      ON    I      7.7;
      O     ;
      A     M     61.5;
      AN    I      0.1;
      =     M     61.5;
NETWORK
TITLE =PROFINET ALARM-모듈이상이나 통신케이블단선(1~10)
//
//
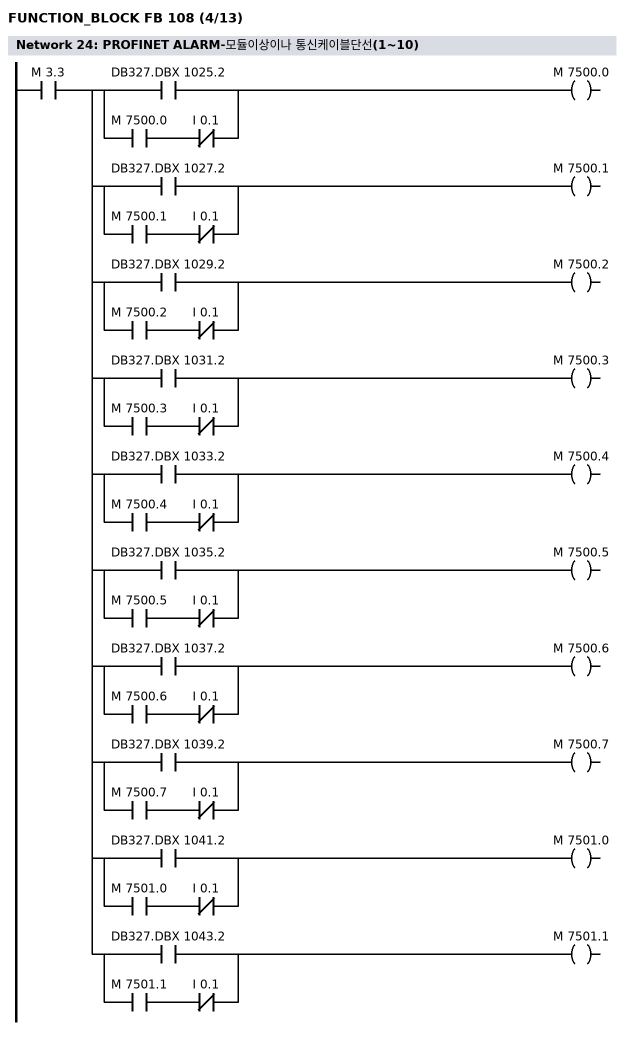
      A     M      3.3;
      =     L      0.0;
      A     L      0.0;
      A(    ;
      O     DB327.DBX 1025.2;
      O     ;
      A     M   7500.0;
      AN    I      0.1;
      )     ;
      =     M   7500.0;
      A     L      0.0;
      A(    ;
      O     DB327.DBX 1027.2;
      O     ;
      A     M   7500.1;
      AN    I      0.1;
      )     ;
      =     M   7500.1;
      A     L      0.0;
      A(    ;
      O     DB327.DBX 1029.2;
      O     ;
      A     M   7500.2;
      AN    I      0.1;
      )     ;
      =     M   7500.2;
      A     L      0.0;
      A(    ;
      O     DB327.DBX 1031.2;
      O     ;
      A     M   7500.3;
      AN    I      0.1;
      )     ;
      =     M   7500.3;
      A     L      0.0;
      A(    ;
      O     DB327.DBX 1033.2;
      O     ;
      A     M   7500.4;
      AN    I      0.1;
      )     ;
      =     M   7500.4;
      A     L      0.0;
      A(    ;
      O     DB327.DBX 1035.2;
      O     ;
      A     M   7500.5;
      AN    I      0.1;
      )     ;
      =     M   7500.5;
      A     L      0.0;
      A(    ;
      O     DB327.DBX 1037.2;
      O     ;
      A     M   7500.6;
      AN    I      0.1;
      )     ;
      =     M   7500.6;
      A     L      0.0;
      A(    ;
      O     DB327.DBX 1039.2;
      O     ;
      A     M   7500.7;
      AN    I      0.1;
      )     ;
      =     M   7500.7;
      A     L      0.0;
      A(    ;
      O     DB327.DBX 1041.2;
      O     ;
      A     M   7501.0;
      AN    I      0.1;
      )     ;
      =     M   7501.0;
      A     L      0.0;
      A(    ;
      O     DB327.DBX 1043.2;
      O     ;
      A     M   7501.1;
      AN    I      0.1;
      )     ;
      =     M   7501.1;
NETWORK
TITLE =PROFINET ALARM-모듈이상이나 통신케이블단선(11~20)
//
//
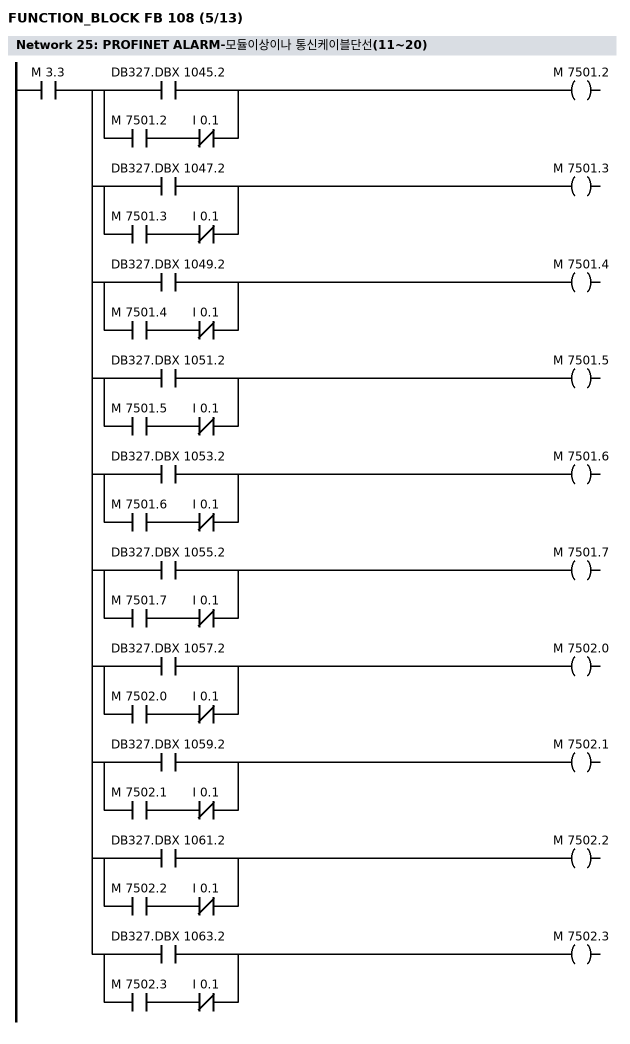
      A     M      3.3;
      =     L      0.0;
      A     L      0.0;
      A(    ;
      O     DB327.DBX 1045.2;
      O     ;
      A     M   7501.2;
      AN    I      0.1;
      )     ;
      =     M   7501.2;
      A     L      0.0;
      A(    ;
      O     DB327.DBX 1047.2;
      O     ;
      A     M   7501.3;
      AN    I      0.1;
      )     ;
      =     M   7501.3;
      A     L      0.0;
      A(    ;
      O     DB327.DBX 1049.2;
      O     ;
      A     M   7501.4;
      AN    I      0.1;
      )     ;
      =     M   7501.4;
      A     L      0.0;
      A(    ;
      O     DB327.DBX 1051.2;
      O     ;
      A     M   7501.5;
      AN    I      0.1;
      )     ;
      =     M   7501.5;
      A     L      0.0;
      A(    ;
      O     DB327.DBX 1053.2;
      O     ;
      A     M   7501.6;
      AN    I      0.1;
      )     ;
      =     M   7501.6;
      A     L      0.0;
      A(    ;
      O     DB327.DBX 1055.2;
      O     ;
      A     M   7501.7;
      AN    I      0.1;
      )     ;
      =     M   7501.7;
      A     L      0.0;
      A(    ;
      O     DB327.DBX 1057.2;
      O     ;
      A     M   7502.0;
      AN    I      0.1;
      )     ;
      =     M   7502.0;
      A     L      0.0;
      A(    ;
      O     DB327.DBX 1059.2;
      O     ;
      A     M   7502.1;
      AN    I      0.1;
      )     ;
      =     M   7502.1;
      A     L      0.0;
      A(    ;
      O     DB327.DBX 1061.2;
      O     ;
      A     M   7502.2;
      AN    I      0.1;
      )     ;
      =     M   7502.2;
      A     L      0.0;
      A(    ;
      O     DB327.DBX 1063.2;
      O     ;
      A     M   7502.3;
      AN    I      0.1;
      )     ;
      =     M   7502.3;
NETWORK
TITLE =PROFINET ALARM-모듈이상이나 통신케이블단선(21~30)
//
//
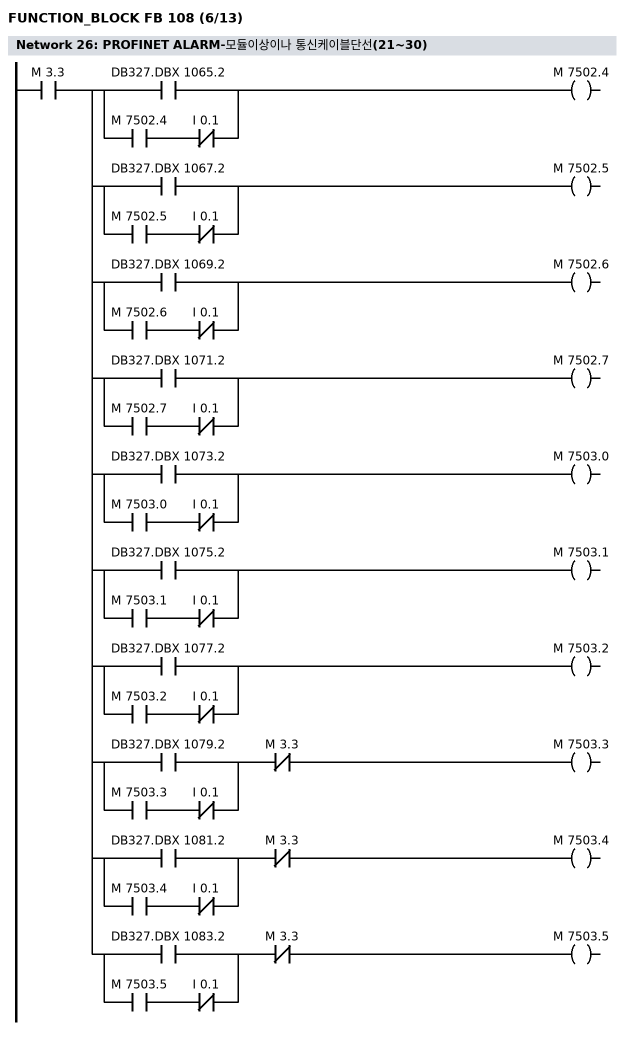
      A     M      3.3;
      =     L      0.0;
      A     L      0.0;
      A(    ;
      O     DB327.DBX 1065.2;
      O     ;
      A     M   7502.4;
      AN    I      0.1;
      )     ;
      =     M   7502.4;
      A     L      0.0;
      A(    ;
      O     DB327.DBX 1067.2;
      O     ;
      A     M   7502.5;
      AN    I      0.1;
      )     ;
      =     M   7502.5;
      A     L      0.0;
      A(    ;
      O     DB327.DBX 1069.2;
      O     ;
      A     M   7502.6;
      AN    I      0.1;
      )     ;
      =     M   7502.6;
      A     L      0.0;
      A(    ;
      O     DB327.DBX 1071.2;
      O     ;
      A     M   7502.7;
      AN    I      0.1;
      )     ;
      =     M   7502.7;
      A     L      0.0;
      A(    ;
      O     DB327.DBX 1073.2;
      O     ;
      A     M   7503.0;
      AN    I      0.1;
      )     ;
      =     M   7503.0;
      A     L      0.0;
      A(    ;
      O     DB327.DBX 1075.2;
      O     ;
      A     M   7503.1;
      AN    I      0.1;
      )     ;
      =     M   7503.1;
      A     L      0.0;
      A(    ;
      O     DB327.DBX 1077.2;
      O     ;
      A     M   7503.2;
      AN    I      0.1;
      )     ;
      =     M   7503.2;
      A     L      0.0;
      A(    ;
      O     DB327.DBX 1079.2;
      O     ;
      A     M   7503.3;
      AN    I      0.1;
      )     ;
      AN    M      3.3;
      =     M   7503.3;
      A     L      0.0;
      A(    ;
      O     DB327.DBX 1081.2;
      O     ;
      A     M   7503.4;
      AN    I      0.1;
      )     ;
      AN    M      3.3;
      =     M   7503.4;
      A     L      0.0;
      A(    ;
      O     DB327.DBX 1083.2;
      O     ;
      A     M   7503.5;
      AN    I      0.1;
      )     ;
      AN    M      3.3;
      =     M   7503.5;
NETWORK
TITLE =PROFINET ALARM-모듈이상이나 통신케이블단선(31~40)
//
//
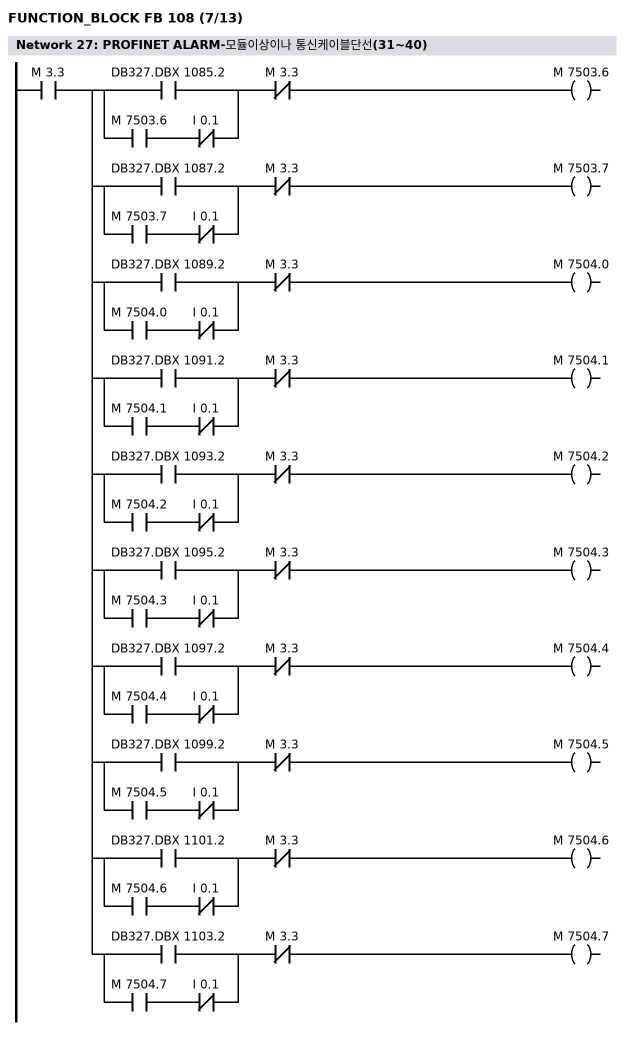
      A     M      3.3;
      =     L      0.0;
      A     L      0.0;
      A(    ;
      O     DB327.DBX 1085.2;
      O     ;
      A     M   7503.6;
      AN    I      0.1;
      )     ;
      AN    M      3.3;
      =     M   7503.6;
      A     L      0.0;
      A(    ;
      O     DB327.DBX 1087.2;
      O     ;
      A     M   7503.7;
      AN    I      0.1;
      )     ;
      AN    M      3.3;
      =     M   7503.7;
      A     L      0.0;
      A(    ;
      O     DB327.DBX 1089.2;
      O     ;
      A     M   7504.0;
      AN    I      0.1;
      )     ;
      AN    M      3.3;
      =     M   7504.0;
      A     L      0.0;
      A(    ;
      O     DB327.DBX 1091.2;
      O     ;
      A     M   7504.1;
      AN    I      0.1;
      )     ;
      AN    M      3.3;
      =     M   7504.1;
      A     L      0.0;
      A(    ;
      O     DB327.DBX 1093.2;
      O     ;
      A     M   7504.2;
      AN    I      0.1;
      )     ;
      AN    M      3.3;
      =     M   7504.2;
      A     L      0.0;
      A(    ;
      O     DB327.DBX 1095.2;
      O     ;
      A     M   7504.3;
      AN    I      0.1;
      )     ;
      AN    M      3.3;
      =     M   7504.3;
      A     L      0.0;
      A(    ;
      O     DB327.DBX 1097.2;
      O     ;
      A     M   7504.4;
      AN    I      0.1;
      )     ;
      AN    M      3.3;
      =     M   7504.4;
      A     L      0.0;
      A(    ;
      O     DB327.DBX 1099.2;
      O     ;
      A     M   7504.5;
      AN    I      0.1;
      )     ;
      AN    M      3.3;
      =     M   7504.5;
      A     L      0.0;
      A(    ;
      O     DB327.DBX 1101.2;
      O     ;
      A     M   7504.6;
      AN    I      0.1;
      )     ;
      AN    M      3.3;
      =     M   7504.6;
      A     L      0.0;
      A(    ;
      O     DB327.DBX 1103.2;
      O     ;
      A     M   7504.7;
      AN    I      0.1;
      )     ;
      AN    M      3.3;
      =     M   7504.7;
NETWORK
TITLE =PROFINET ALARM-모듈이상이나 통신케이블단선(150~159)
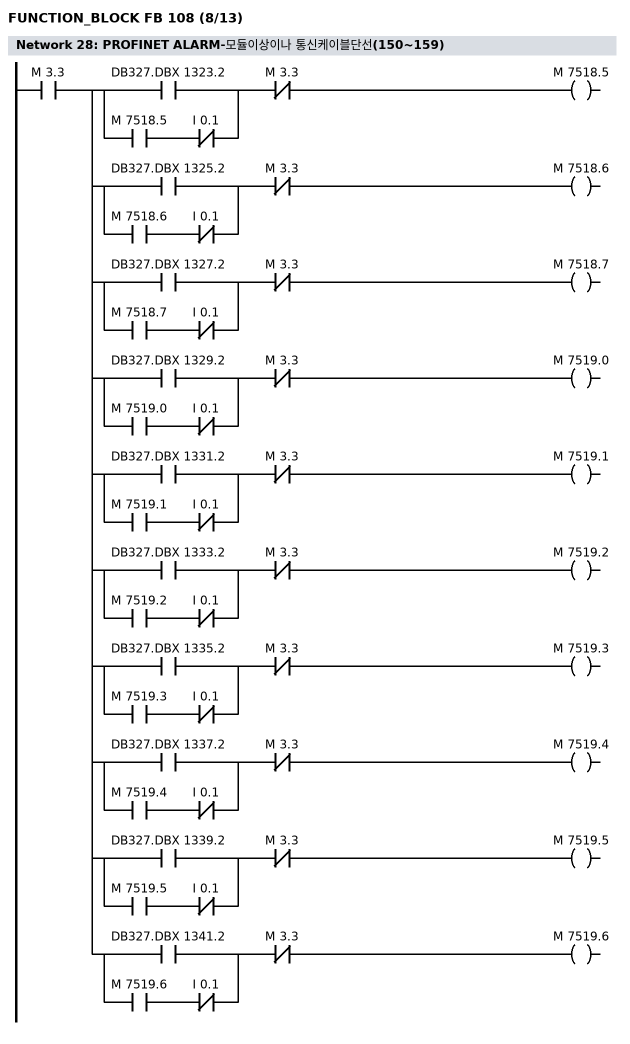

      A     M      3.3;
      =     L      0.0;
      A     L      0.0;
      A(    ;
      O     DB327.DBX 1323.2;
      O     ;
      A     M   7518.5;
      AN    I      0.1;
      )     ;
      AN    M      3.3;
      =     M   7518.5;
      A     L      0.0;
      A(    ;
      O     DB327.DBX 1325.2;
      O     ;
      A     M   7518.6;
      AN    I      0.1;
      )     ;
      AN    M      3.3;
      =     M   7518.6;
      A     L      0.0;
      A(    ;
      O     DB327.DBX 1327.2;
      O     ;
      A     M   7518.7;
      AN    I      0.1;
      )     ;
      AN    M      3.3;
      =     M   7518.7;
      A     L      0.0;
      A(    ;
      O     DB327.DBX 1329.2;
      O     ;
      A     M   7519.0;
      AN    I      0.1;
      )     ;
      AN    M      3.3;
      =     M   7519.0;
      A     L      0.0;
      A(    ;
      O     DB327.DBX 1331.2;
      O     ;
      A     M   7519.1;
      AN    I      0.1;
      )     ;
      AN    M      3.3;
      =     M   7519.1;
      A     L      0.0;
      A(    ;
      O     DB327.DBX 1333.2;
      O     ;
      A     M   7519.2;
      AN    I      0.1;
      )     ;
      AN    M      3.3;
      =     M   7519.2;
      A     L      0.0;
      A(    ;
      O     DB327.DBX 1335.2;
      O     ;
      A     M   7519.3;
      AN    I      0.1;
      )     ;
      AN    M      3.3;
      =     M   7519.3;
      A     L      0.0;
      A(    ;
      O     DB327.DBX 1337.2;
      O     ;
      A     M   7519.4;
      AN    I      0.1;
      )     ;
      AN    M      3.3;
      =     M   7519.4;
      A     L      0.0;
      A(    ;
      O     DB327.DBX 1339.2;
      O     ;
      A     M   7519.5;
      AN    I      0.1;
      )     ;
      AN    M      3.3;
      =     M   7519.5;
      A     L      0.0;
      A(    ;
      O     DB327.DBX 1341.2;
      O     ;
      A     M   7519.6;
      AN    I      0.1;
      )     ;
      AN    M      3.3;
      =     M   7519.6;
NETWORK
TITLE =PROFINET MODULE ERROR(1~10)
//
//
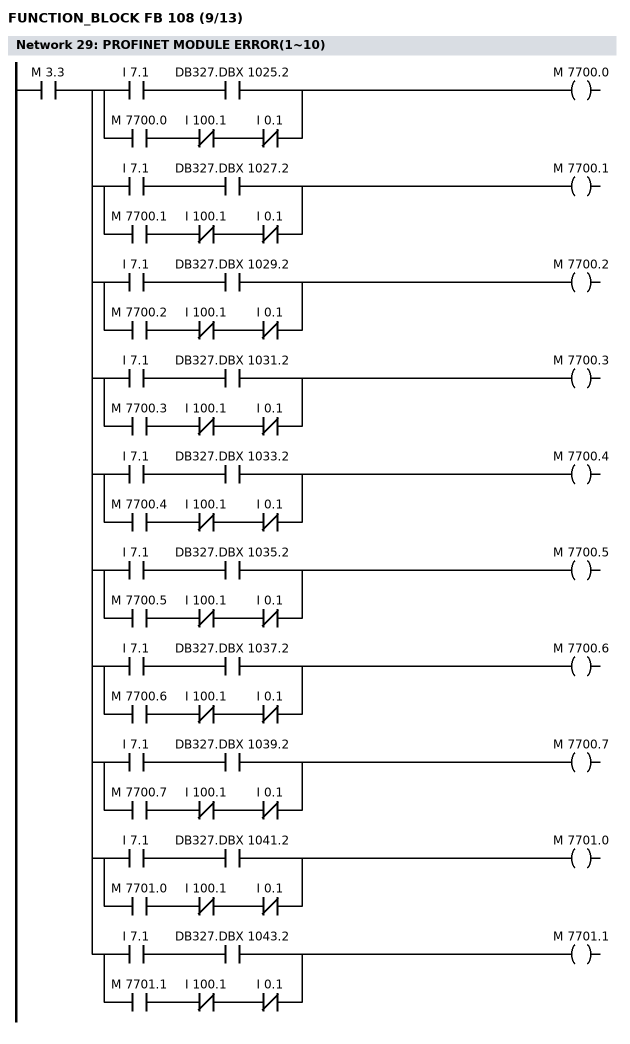
      A     M      3.3;
      =     L      0.0;
      A     L      0.0;
      A(    ;
      A     I      7.1;
      A     DB327.DBX 1025.2;
      O     ;
      A     M   7700.0;
      AN    I    100.1;
      AN    I      0.1;
      )     ;
      =     M   7700.0;
      A     L      0.0;
      A(    ;
      A     I      7.1;
      A     DB327.DBX 1027.2;
      O     ;
      A     M   7700.1;
      AN    I    100.1;
      AN    I      0.1;
      )     ;
      =     M   7700.1;
      A     L      0.0;
      A(    ;
      A     I      7.1;
      A     DB327.DBX 1029.2;
      O     ;
      A     M   7700.2;
      AN    I    100.1;
      AN    I      0.1;
      )     ;
      =     M   7700.2;
      A     L      0.0;
      A(    ;
      A     I      7.1;
      A     DB327.DBX 1031.2;
      O     ;
      A     M   7700.3;
      AN    I    100.1;
      AN    I      0.1;
      )     ;
      =     M   7700.3;
      A     L      0.0;
      A(    ;
      A     I      7.1;
      A     DB327.DBX 1033.2;
      O     ;
      A     M   7700.4;
      AN    I    100.1;
      AN    I      0.1;
      )     ;
      =     M   7700.4;
      A     L      0.0;
      A(    ;
      A     I      7.1;
      A     DB327.DBX 1035.2;
      O     ;
      A     M   7700.5;
      AN    I    100.1;
      AN    I      0.1;
      )     ;
      =     M   7700.5;
      A     L      0.0;
      A(    ;
      A     I      7.1;
      A     DB327.DBX 1037.2;
      O     ;
      A     M   7700.6;
      AN    I    100.1;
      AN    I      0.1;
      )     ;
      =     M   7700.6;
      A     L      0.0;
      A(    ;
      A     I      7.1;
      A     DB327.DBX 1039.2;
      O     ;
      A     M   7700.7;
      AN    I    100.1;
      AN    I      0.1;
      )     ;
      =     M   7700.7;
      A     L      0.0;
      A(    ;
      A     I      7.1;
      A     DB327.DBX 1041.2;
      O     ;
      A     M   7701.0;
      AN    I    100.1;
      AN    I      0.1;
      )     ;
      =     M   7701.0;
      A     L      0.0;
      A(    ;
      A     I      7.1;
      A     DB327.DBX 1043.2;
      O     ;
      A     M   7701.1;
      AN    I    100.1;
      AN    I      0.1;
      )     ;
      =     M   7701.1;
NETWORK
TITLE =PROFINET MODULE ERROR(11~20)
//
//
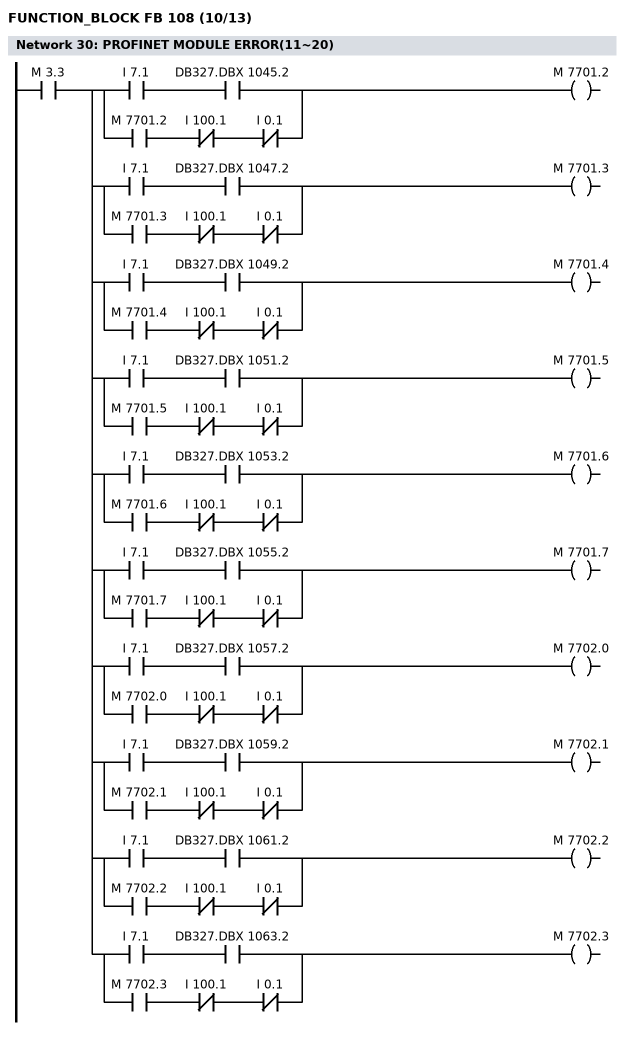
      A     M      3.3;
      =     L      0.0;
      A     L      0.0;
      A(    ;
      A     I      7.1;
      A     DB327.DBX 1045.2;
      O     ;
      A     M   7701.2;
      AN    I    100.1;
      AN    I      0.1;
      )     ;
      =     M   7701.2;
      A     L      0.0;
      A(    ;
      A     I      7.1;
      A     DB327.DBX 1047.2;
      O     ;
      A     M   7701.3;
      AN    I    100.1;
      AN    I      0.1;
      )     ;
      =     M   7701.3;
      A     L      0.0;
      A(    ;
      A     I      7.1;
      A     DB327.DBX 1049.2;
      O     ;
      A     M   7701.4;
      AN    I    100.1;
      AN    I      0.1;
      )     ;
      =     M   7701.4;
      A     L      0.0;
      A(    ;
      A     I      7.1;
      A     DB327.DBX 1051.2;
      O     ;
      A     M   7701.5;
      AN    I    100.1;
      AN    I      0.1;
      )     ;
      =     M   7701.5;
      A     L      0.0;
      A(    ;
      A     I      7.1;
      A     DB327.DBX 1053.2;
      O     ;
      A     M   7701.6;
      AN    I    100.1;
      AN    I      0.1;
      )     ;
      =     M   7701.6;
      A     L      0.0;
      A(    ;
      A     I      7.1;
      A     DB327.DBX 1055.2;
      O     ;
      A     M   7701.7;
      AN    I    100.1;
      AN    I      0.1;
      )     ;
      =     M   7701.7;
      A     L      0.0;
      A(    ;
      A     I      7.1;
      A     DB327.DBX 1057.2;
      O     ;
      A     M   7702.0;
      AN    I    100.1;
      AN    I      0.1;
      )     ;
      =     M   7702.0;
      A     L      0.0;
      A(    ;
      A     I      7.1;
      A     DB327.DBX 1059.2;
      O     ;
      A     M   7702.1;
      AN    I    100.1;
      AN    I      0.1;
      )     ;
      =     M   7702.1;
      A     L      0.0;
      A(    ;
      A     I      7.1;
      A     DB327.DBX 1061.2;
      O     ;
      A     M   7702.2;
      AN    I    100.1;
      AN    I      0.1;
      )     ;
      =     M   7702.2;
      A     L      0.0;
      A(    ;
      A     I      7.1;
      A     DB327.DBX 1063.2;
      O     ;
      A     M   7702.3;
      AN    I    100.1;
      AN    I      0.1;
      )     ;
      =     M   7702.3;
NETWORK
TITLE =PROFINET MODULE ERROR(21~30)
//
//
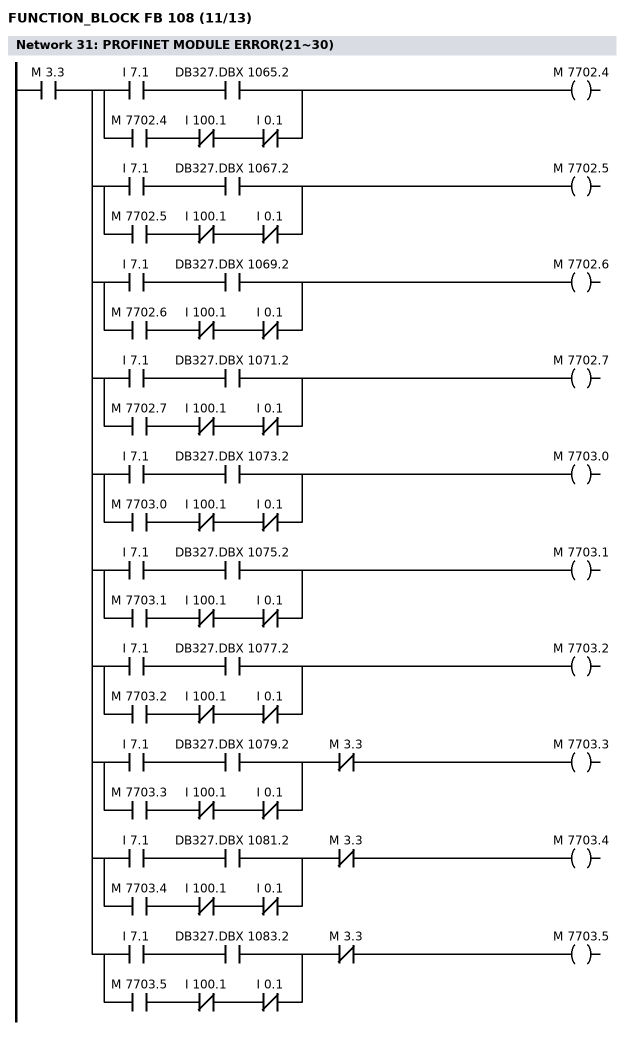
      A     M      3.3;
      =     L      0.0;
      A     L      0.0;
      A(    ;
      A     I      7.1;
      A     DB327.DBX 1065.2;
      O     ;
      A     M   7702.4;
      AN    I    100.1;
      AN    I      0.1;
      )     ;
      =     M   7702.4;
      A     L      0.0;
      A(    ;
      A     I      7.1;
      A     DB327.DBX 1067.2;
      O     ;
      A     M   7702.5;
      AN    I    100.1;
      AN    I      0.1;
      )     ;
      =     M   7702.5;
      A     L      0.0;
      A(    ;
      A     I      7.1;
      A     DB327.DBX 1069.2;
      O     ;
      A     M   7702.6;
      AN    I    100.1;
      AN    I      0.1;
      )     ;
      =     M   7702.6;
      A     L      0.0;
      A(    ;
      A     I      7.1;
      A     DB327.DBX 1071.2;
      O     ;
      A     M   7702.7;
      AN    I    100.1;
      AN    I      0.1;
      )     ;
      =     M   7702.7;
      A     L      0.0;
      A(    ;
      A     I      7.1;
      A     DB327.DBX 1073.2;
      O     ;
      A     M   7703.0;
      AN    I    100.1;
      AN    I      0.1;
      )     ;
      =     M   7703.0;
      A     L      0.0;
      A(    ;
      A     I      7.1;
      A     DB327.DBX 1075.2;
      O     ;
      A     M   7703.1;
      AN    I    100.1;
      AN    I      0.1;
      )     ;
      =     M   7703.1;
      A     L      0.0;
      A(    ;
      A     I      7.1;
      A     DB327.DBX 1077.2;
      O     ;
      A     M   7703.2;
      AN    I    100.1;
      AN    I      0.1;
      )     ;
      =     M   7703.2;
      A     L      0.0;
      A(    ;
      A     I      7.1;
      A     DB327.DBX 1079.2;
      O     ;
      A     M   7703.3;
      AN    I    100.1;
      AN    I      0.1;
      )     ;
      AN    M      3.3;
      =     M   7703.3;
      A     L      0.0;
      A(    ;
      A     I      7.1;
      A     DB327.DBX 1081.2;
      O     ;
      A     M   7703.4;
      AN    I    100.1;
      AN    I      0.1;
      )     ;
      AN    M      3.3;
      =     M   7703.4;
      A     L      0.0;
      A(    ;
      A     I      7.1;
      A     DB327.DBX 1083.2;
      O     ;
      A     M   7703.5;
      AN    I    100.1;
      AN    I      0.1;
      )     ;
      AN    M      3.3;
      =     M   7703.5;
NETWORK
TITLE =PROFINET MODULE ERROR(31~40)
//
//
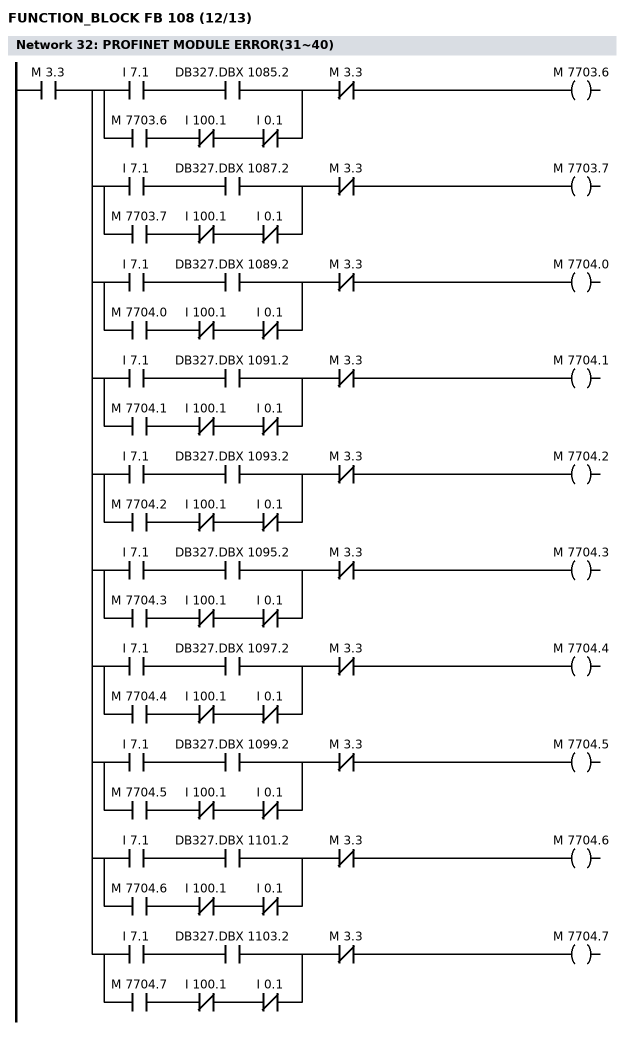
      A     M      3.3;
      =     L      0.0;
      A     L      0.0;
      A(    ;
      A     I      7.1;
      A     DB327.DBX 1085.2;
      O     ;
      A     M   7703.6;
      AN    I    100.1;
      AN    I      0.1;
      )     ;
      AN    M      3.3;
      =     M   7703.6;
      A     L      0.0;
      A(    ;
      A     I      7.1;
      A     DB327.DBX 1087.2;
      O     ;
      A     M   7703.7;
      AN    I    100.1;
      AN    I      0.1;
      )     ;
      AN    M      3.3;
      =     M   7703.7;
      A     L      0.0;
      A(    ;
      A     I      7.1;
      A     DB327.DBX 1089.2;
      O     ;
      A     M   7704.0;
      AN    I    100.1;
      AN    I      0.1;
      )     ;
      AN    M      3.3;
      =     M   7704.0;
      A     L      0.0;
      A(    ;
      A     I      7.1;
      A     DB327.DBX 1091.2;
      O     ;
      A     M   7704.1;
      AN    I    100.1;
      AN    I      0.1;
      )     ;
      AN    M      3.3;
      =     M   7704.1;
      A     L      0.0;
      A(    ;
      A     I      7.1;
      A     DB327.DBX 1093.2;
      O     ;
      A     M   7704.2;
      AN    I    100.1;
      AN    I      0.1;
      )     ;
      AN    M      3.3;
      =     M   7704.2;
      A     L      0.0;
      A(    ;
      A     I      7.1;
      A     DB327.DBX 1095.2;
      O     ;
      A     M   7704.3;
      AN    I    100.1;
      AN    I      0.1;
      )     ;
      AN    M      3.3;
      =     M   7704.3;
      A     L      0.0;
      A(    ;
      A     I      7.1;
      A     DB327.DBX 1097.2;
      O     ;
      A     M   7704.4;
      AN    I    100.1;
      AN    I      0.1;
      )     ;
      AN    M      3.3;
      =     M   7704.4;
      A     L      0.0;
      A(    ;
      A     I      7.1;
      A     DB327.DBX 1099.2;
      O     ;
      A     M   7704.5;
      AN    I    100.1;
      AN    I      0.1;
      )     ;
      AN    M      3.3;
      =     M   7704.5;
      A     L      0.0;
      A(    ;
      A     I      7.1;
      A     DB327.DBX 1101.2;
      O     ;
      A     M   7704.6;
      AN    I    100.1;
      AN    I      0.1;
      )     ;
      AN    M      3.3;
      =     M   7704.6;
      A     L      0.0;
      A(    ;
      A     I      7.1;
      A     DB327.DBX 1103.2;
      O     ;
      A     M   7704.7;
      AN    I    100.1;
      AN    I      0.1;
      )     ;
      AN    M      3.3;
      =     M   7704.7;
NETWORK
TITLE =PROFINET MODULE ERROR(150~159)
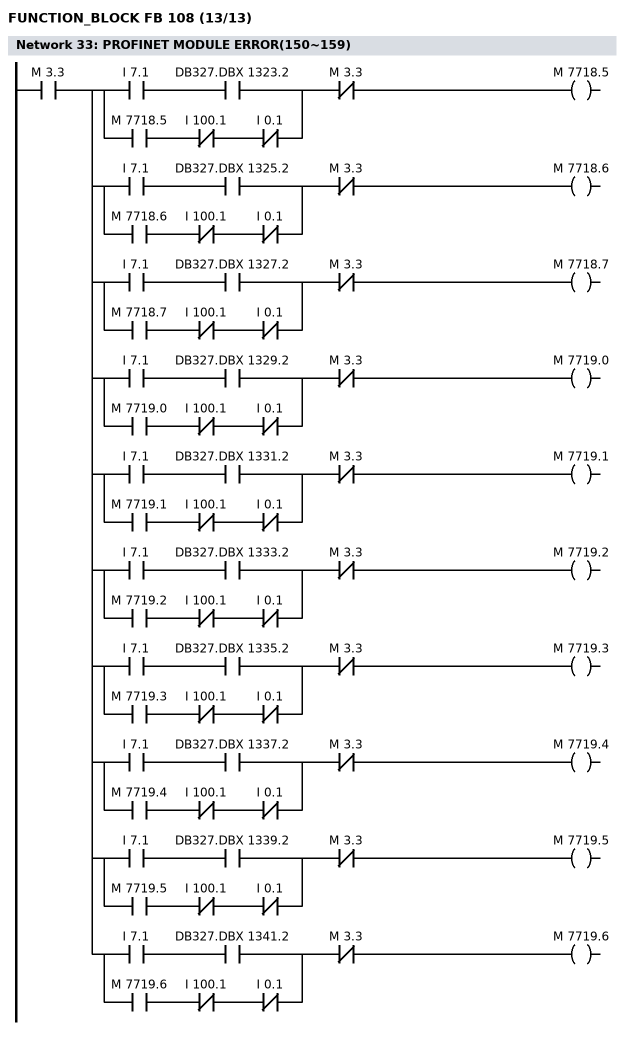

      A     M      3.3;
      =     L      0.0;
      A     L      0.0;
      A(    ;
      A     I      7.1;
      A     DB327.DBX 1323.2;
      O     ;
      A     M   7718.5;
      AN    I    100.1;
      AN    I      0.1;
      )     ;
      AN    M      3.3;
      =     M   7718.5;
      A     L      0.0;
      A(    ;
      A     I      7.1;
      A     DB327.DBX 1325.2;
      O     ;
      A     M   7718.6;
      AN    I    100.1;
      AN    I      0.1;
      )     ;
      AN    M      3.3;
      =     M   7718.6;
      A     L      0.0;
      A(    ;
      A     I      7.1;
      A     DB327.DBX 1327.2;
      O     ;
      A     M   7718.7;
      AN    I    100.1;
      AN    I      0.1;
      )     ;
      AN    M      3.3;
      =     M   7718.7;
      A     L      0.0;
      A(    ;
      A     I      7.1;
      A     DB327.DBX 1329.2;
      O     ;
      A     M   7719.0;
      AN    I    100.1;
      AN    I      0.1;
      )     ;
      AN    M      3.3;
      =     M   7719.0;
      A     L      0.0;
      A(    ;
      A     I      7.1;
      A     DB327.DBX 1331.2;
      O     ;
      A     M   7719.1;
      AN    I    100.1;
      AN    I      0.1;
      )     ;
      AN    M      3.3;
      =     M   7719.1;
      A     L      0.0;
      A(    ;
      A     I      7.1;
      A     DB327.DBX 1333.2;
      O     ;
      A     M   7719.2;
      AN    I    100.1;
      AN    I      0.1;
      )     ;
      AN    M      3.3;
      =     M   7719.2;
      A     L      0.0;
      A(    ;
      A     I      7.1;
      A     DB327.DBX 1335.2;
      O     ;
      A     M   7719.3;
      AN    I    100.1;
      AN    I      0.1;
      )     ;
      AN    M      3.3;
      =     M   7719.3;
      A     L      0.0;
      A(    ;
      A     I      7.1;
      A     DB327.DBX 1337.2;
      O     ;
      A     M   7719.4;
      AN    I    100.1;
      AN    I      0.1;
      )     ;
      AN    M      3.3;
      =     M   7719.4;
      A     L      0.0;
      A(    ;
      A     I      7.1;
      A     DB327.DBX 1339.2;
      O     ;
      A     M   7719.5;
      AN    I    100.1;
      AN    I      0.1;
      )     ;
      AN    M      3.3;
      =     M   7719.5;
      A     L      0.0;
      A(    ;
      A     I      7.1;
      A     DB327.DBX 1341.2;
      O     ;
      A     M   7719.6;
      AN    I    100.1;
      AN    I      0.1;
      )     ;
      AN    M      3.3;
      =     M   7719.6;
END_FUNCTION_BLOCK

DATA_BLOCK DB 108
TITLE =
VERSION : 0.0

 FB 108
BEGIN
END_DATA_BLOCK

FUNCTION_BLOCK FB 110
TITLE =
VERSION : 0.1


VAR
  S711A_MODE : FB 402;
  S711B_MODE : FB 402;
END_VAR
BEGIN
NETWORK
TITLE =
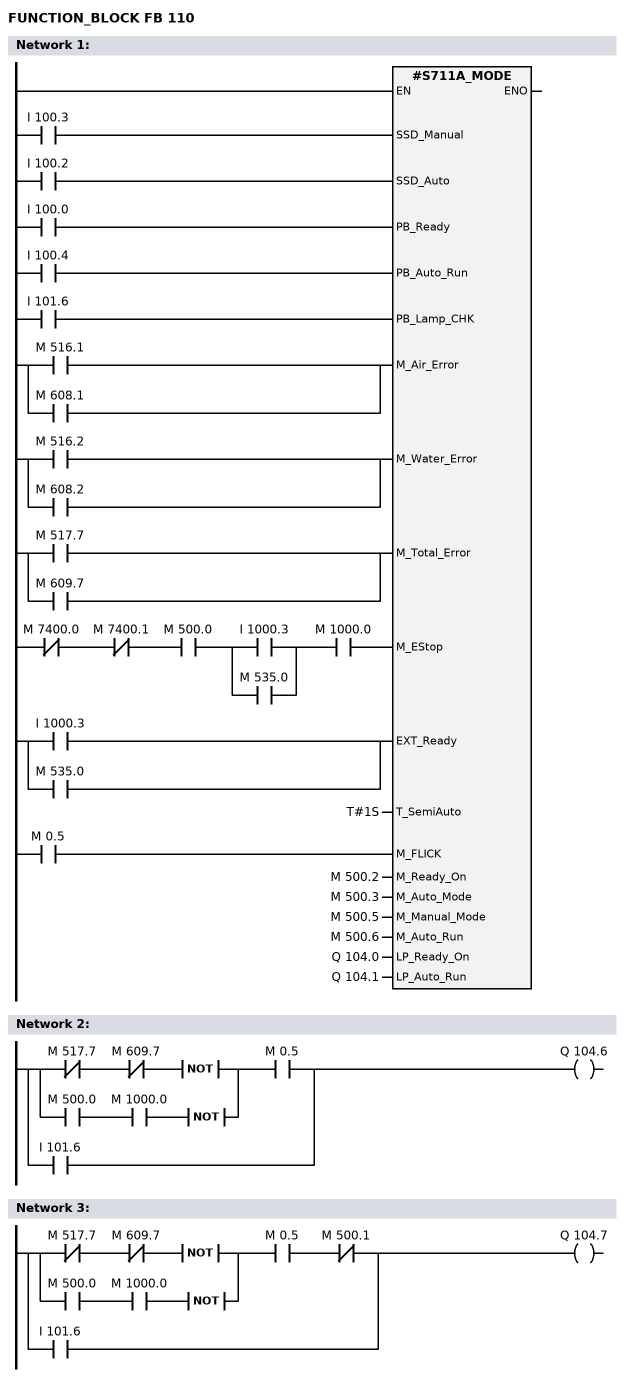

      A     I    100.3;
      =     L      0.0;
      BLD   103;
      A     I    100.2;
      =     L      0.1;
      BLD   103;
      A     I    100.0;
      =     L      0.2;
      BLD   103;
      A     I    100.4;
      =     L      0.3;
      BLD   103;
      A     I    101.6;
      =     L      0.6;
      BLD   103;
      A(    ;
      O     M    516.1;
      O     M    608.1;
      )     ;
      =     L      0.7;
      BLD   103;
      A(    ;
      O     M    516.2;
      O     M    608.2;
      )     ;
      =     L      1.0;
      BLD   103;
      A(    ;
      O     M    517.7;
      O     M    609.7;
      )     ;
      =     L      1.1;
      BLD   103;
      AN    M   7400.0;
      AN    M   7400.1;
      A     M    500.0;
      A(    ;
      O     I   1000.3;
      O     M    535.0;
      )     ;
      A     M   1000.0;
      =     L      1.2;
      BLD   103;
      A(    ;
      O     I   1000.3;
      O     M    535.0;
      )     ;
      =     L      1.3;
      BLD   103;
      A     M      0.5;
      =     L      1.5;
      BLD   103;
      CALL #S711A_MODE (
           SSD_Manual               := L      0.0,
           SSD_Auto                 := L      0.1,
           PB_Ready                 := L      0.2,
           PB_Auto_Run              := L      0.3,
           PB_Lamp_CHK              := L      0.6,
           M_Air_Error              := L      0.7,
           M_Water_Error            := L      1.0,
           M_Total_Error            := L      1.1,
           M_EStop                  := L      1.2,
           EXT_Ready                := L      1.3,
           T_SemiAuto               := T#1S,
           M_FLICK                  := L      1.5,
           M_Ready_On               := M    500.2,
           M_Auto_Mode              := M    500.3,
           M_Manual_Mode            := M    500.5,
           M_Auto_Run               := M    500.6,
           LP_Ready_On              := Q    104.0,
           LP_Auto_Run              := Q    104.1);
      NOP   0;
NETWORK
TITLE =

      A(    ;
      AN    M    517.7;
      AN    M    609.7;
      NOT   ;
      O(    ;
      A     M    500.0;
      A     M   1000.0;
      NOT   ;
      )     ;
      )     ;
      A     M      0.5;
      O     I    101.6;
      =     Q    104.6;
NETWORK
TITLE =

      A(    ;
      AN    M    517.7;
      AN    M    609.7;
      NOT   ;
      O(    ;
      A     M    500.0;
      A     M   1000.0;
      NOT   ;
      )     ;
      )     ;
      A     M      0.5;
      AN    M    500.1;
      O     I    101.6;
      =     Q    104.7;
NETWORK
TITLE =보조조작반 램프

      AN    OV;
      =     L      0.0;
      A     L      0.0;
      A     M    501.0;
      =     Q     51.7;
      A     L      0.0;
      AN    I     43.4;
      =     Q     51.6;
      A     L      0.0;
      A     M    600.1;
      =     Q     51.5;
END_FUNCTION_BLOCK

DATA_BLOCK DB 110
TITLE =
VERSION : 0.0

 FB 110
BEGIN
   S711A_MODE.SSD_Manual := FALSE;
   S711A_MODE.SSD_Auto := FALSE;
   S711A_MODE.PB_Ready := FALSE;
   S711A_MODE.PB_Auto_Run := FALSE;
   S711A_MODE.PB_Remote_Ready := FALSE;
   S711A_MODE.PB_Remote_Auto_Run := FALSE;
   S711A_MODE.PB_Lamp_CHK := FALSE;
   S711A_MODE.M_Air_Error := FALSE;
   S711A_MODE.M_Water_Error := FALSE;
   S711A_MODE.M_Total_Error := FALSE;
   S711A_MODE.M_EStop := FALSE;
   S711A_MODE.EXT_Ready := FALSE;
   S711A_MODE.EXT_Auto := FALSE;
   S711A_MODE.T_SemiAuto := T#0MS;
   S711A_MODE.M_FLICK := FALSE;
   S711A_MODE.M_Ready_On := FALSE;
   S711A_MODE.M_Auto_Mode := FALSE;
   S711A_MODE.M_SemiAuto_Mode := FALSE;
   S711A_MODE.M_Manual_Mode := FALSE;
   S711A_MODE.M_Auto_Run := FALSE;
   S711A_MODE.LP_Ready_On := FALSE;
   S711A_MODE.LP_Auto_Run := FALSE;
   S711A_MODE.AUTO_MODE_DELAY.IN := FALSE;
   S711A_MODE.AUTO_MODE_DELAY.PT := T#0MS;
   S711A_MODE.AUTO_MODE_DELAY.Q := FALSE;
   S711A_MODE.AUTO_MODE_DELAY.ET := T#0MS;
   S711A_MODE.AUTO_MODE_DELAY.STATE := B#16#0;
   S711A_MODE.AUTO_MODE_DELAY.STIME := T#0MS;
   S711A_MODE.AUTO_MODE_DELAY.ATIME := T#0MS;
   S711A_MODE.SEMI_AUTO_DELAY.IN := FALSE;
   S711A_MODE.SEMI_AUTO_DELAY.PT := T#0MS;
   S711A_MODE.SEMI_AUTO_DELAY.Q := FALSE;
   S711A_MODE.SEMI_AUTO_DELAY.ET := T#0MS;
   S711A_MODE.SEMI_AUTO_DELAY.STATE := B#16#0;
   S711A_MODE.SEMI_AUTO_DELAY.STIME := T#0MS;
   S711A_MODE.SEMI_AUTO_DELAY.ATIME := T#0MS;
   S711A_MODE.MANUAL_DELAY.IN := FALSE;
   S711A_MODE.MANUAL_DELAY.PT := T#0MS;
   S711A_MODE.MANUAL_DELAY.Q := FALSE;
   S711A_MODE.MANUAL_DELAY.ET := T#0MS;
   S711A_MODE.MANUAL_DELAY.STATE := B#16#0;
   S711A_MODE.MANUAL_DELAY.STIME := T#0MS;
   S711A_MODE.MANUAL_DELAY.ATIME := T#0MS;
   S711B_MODE.SSD_Manual := FALSE;
   S711B_MODE.SSD_Auto := FALSE;
   S711B_MODE.PB_Ready := FALSE;
   S711B_MODE.PB_Auto_Run := FALSE;
   S711B_MODE.PB_Remote_Ready := FALSE;
   S711B_MODE.PB_Remote_Auto_Run := FALSE;
   S711B_MODE.PB_Lamp_CHK := FALSE;
   S711B_MODE.M_Air_Error := FALSE;
   S711B_MODE.M_Water_Error := FALSE;
   S711B_MODE.M_Total_Error := FALSE;
   S711B_MODE.M_EStop := FALSE;
   S711B_MODE.EXT_Ready := FALSE;
   S711B_MODE.EXT_Auto := FALSE;
   S711B_MODE.T_SemiAuto := T#0MS;
   S711B_MODE.M_FLICK := FALSE;
   S711B_MODE.M_Ready_On := FALSE;
   S711B_MODE.M_Auto_Mode := FALSE;
   S711B_MODE.M_SemiAuto_Mode := FALSE;
   S711B_MODE.M_Manual_Mode := FALSE;
   S711B_MODE.M_Auto_Run := FALSE;
   S711B_MODE.LP_Ready_On := FALSE;
   S711B_MODE.LP_Auto_Run := FALSE;
   S711B_MODE.AUTO_MODE_DELAY.IN := FALSE;
   S711B_MODE.AUTO_MODE_DELAY.PT := T#0MS;
   S711B_MODE.AUTO_MODE_DELAY.Q := FALSE;
   S711B_MODE.AUTO_MODE_DELAY.ET := T#0MS;
   S711B_MODE.AUTO_MODE_DELAY.STATE := B#16#0;
   S711B_MODE.AUTO_MODE_DELAY.STIME := T#0MS;
   S711B_MODE.AUTO_MODE_DELAY.ATIME := T#0MS;
   S711B_MODE.SEMI_AUTO_DELAY.IN := FALSE;
   S711B_MODE.SEMI_AUTO_DELAY.PT := T#0MS;
   S711B_MODE.SEMI_AUTO_DELAY.Q := FALSE;
   S711B_MODE.SEMI_AUTO_DELAY.ET := T#0MS;
   S711B_MODE.SEMI_AUTO_DELAY.STATE := B#16#0;
   S711B_MODE.SEMI_AUTO_DELAY.STIME := T#0MS;
   S711B_MODE.SEMI_AUTO_DELAY.ATIME := T#0MS;
   S711B_MODE.MANUAL_DELAY.IN := FALSE;
   S711B_MODE.MANUAL_DELAY.PT := T#0MS;
   S711B_MODE.MANUAL_DELAY.Q := FALSE;
   S711B_MODE.MANUAL_DELAY.ET := T#0MS;
   S711B_MODE.MANUAL_DELAY.STATE := B#16#0;
   S711B_MODE.MANUAL_DELAY.STIME := T#0MS;
   S711B_MODE.MANUAL_DELAY.ATIME := T#0MS;
END_DATA_BLOCK

FUNCTION FC 110 : VOID
TITLE =
VERSION : 0.1

BEGIN
NETWORK
TITLE =
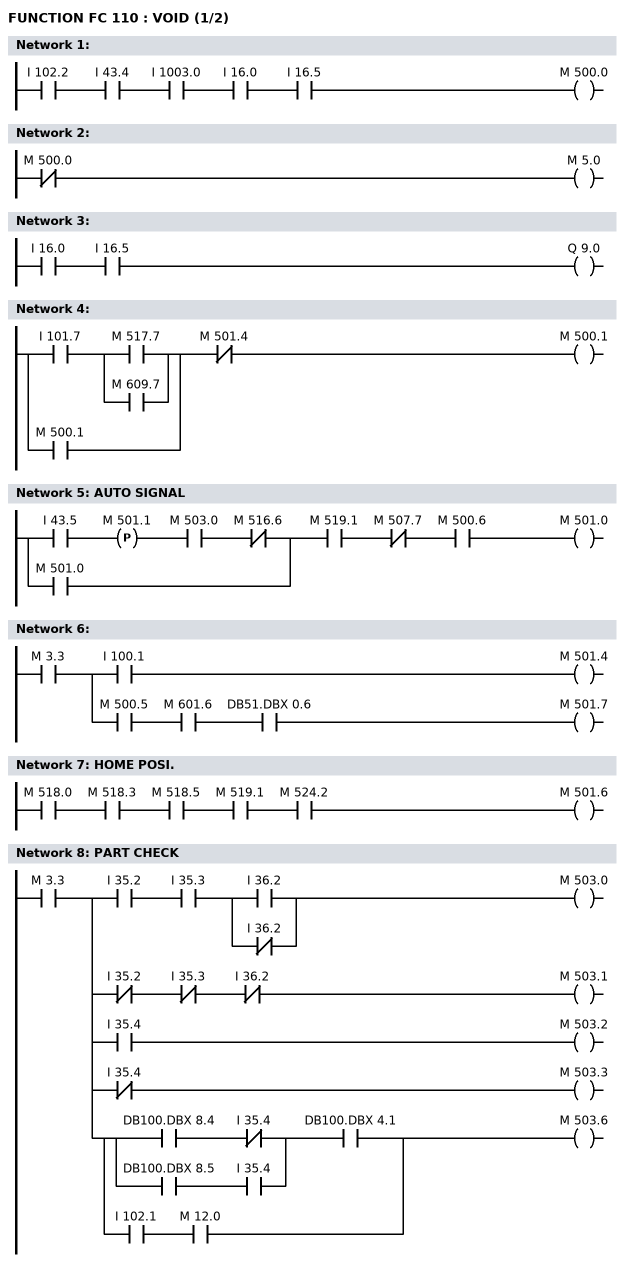

      A     I    102.2;
      A     I     43.4;
      A     I   1003.0;
      A     I     16.0;
      A     I     16.5;
      =     M    500.0;
NETWORK
TITLE =

      AN    M    500.0;
      =     M      5.0;
NETWORK
TITLE =

      A     I     16.0;
      A     I     16.5;
      =     Q      9.0;
NETWORK
TITLE =

      A(    ;
      A     I    101.7;
      A(    ;
      O     M    517.7;
      O     M    609.7;
      )     ;
      O     M    500.1;
      )     ;
      AN    M    501.4;
      =     M    500.1;
NETWORK
TITLE =AUTO SIGNAL

      A(    ;
      A     I     43.5;
      FP    M    501.1;
      A     M    503.0;
      AN    M    516.6;
      O     M    501.0;
      )     ;
      A     M    519.1;
      AN    M    507.7;
      A     M    500.6;
      =     M    501.0;
NETWORK
TITLE =

      A     M      3.3;
      =     L      0.0;
      A     L      0.0;
      A     I    100.1;
      =     M    501.4;
      A     L      0.0;
      A     M    500.5;
      A     M    601.6;
      A     DB51.DBX    0.6;
      =     M    501.7;
NETWORK
TITLE =HOME POSI.

      A     M    518.0;
      A     M    518.3;
      A     M    518.5;
      A     M    519.1;
      A     M    524.2;
      =     M    501.6;
NETWORK
TITLE =PART CHECK

      A     M      3.3;
      =     L      0.0;
      A     L      0.0;
      A     I     35.2;
      A     I     35.3;
      A(    ;
      O     I     36.2;
      ON    I     36.2;
      )     ;
      =     M    503.0;
      A     L      0.0;
      AN    I     35.2;
      AN    I     35.3;
      AN    I     36.2;
      =     M    503.1;
      A     L      0.0;
      A     I     35.4;
      =     M    503.2;
      A     L      0.0;
      AN    I     35.4;
      =     M    503.3;
      A     L      0.0;
      A(    ;
      A(    ;
      A     DB100.DBX    8.4;
      AN    I     35.4;
      O     ;
      A     DB100.DBX    8.5;
      A     I     35.4;
      )     ;
      A     DB100.DBX    4.1;
      O     ;
      A     I    102.1;
      A     M     12.0;
      )     ;
      =     M    503.6;
NETWORK
TITLE =
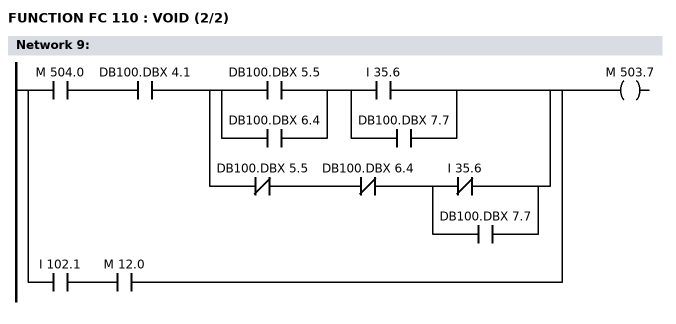

      A     M    504.0;
      A     DB100.DBX    4.1;
      A(    ;
      A(    ;
      O     DB100.DBX    5.5;
      O     DB100.DBX    6.4;
      )     ;
      A(    ;
      O     I     35.6;
      O     DB100.DBX    7.7;
      )     ;
      O     ;
      AN    DB100.DBX    5.5;
      AN    DB100.DBX    6.4;
      A(    ;
      ON    I     35.6;
      O     DB100.DBX    7.7;
      )     ;
      )     ;
      O     ;
      A     I    102.1;
      A     M     12.0;
      =     M    503.7;
NETWORK
TITLE =CAM1 UP ACTION

      A     M    500.5;
      =     L      0.0;
      A     L      0.0;
      A     M    601.6;
      =     L      0.1;
      A     L      0.1;
      AN    DB51.DBX    3.7;
      A     DB51.DBX    3.6;
      =     M    511.6;
      A     L      0.1;
      A     DB51.DBX    3.7;
      AN    DB51.DBX    3.6;
      =     M    511.7;
      A     L      0.0;
      A     M    601.7;
      =     L      0.1;
      A     L      0.1;
      AN    DB51.DBX    3.7;
      A     DB51.DBX    3.6;
      =     M    603.6;
      A     L      0.1;
      A     DB51.DBX    3.7;
      AN    DB51.DBX    3.6;
      =     M    603.7;
NETWORK
TITLE =

      AN    OV;
      =     L      0.0;
      A     L      0.0;
      A(    ;
      O     I   1002.5;
      O     I   1000.0;
      O     I   1000.7;
      )     ;
      =     M    530.4;
      A     L      0.0;
      A(    ;
      O     I   1002.6;
      O     I   1000.0;
      O     I   1000.7;
      )     ;
      =     M    530.5;
      A     L      0.0;
      A(    ;
      O     I   1002.7;
      O     I   1000.0;
      O     I   1000.7;
      )     ;
      =     M    530.6;
NETWORK
TITLE =
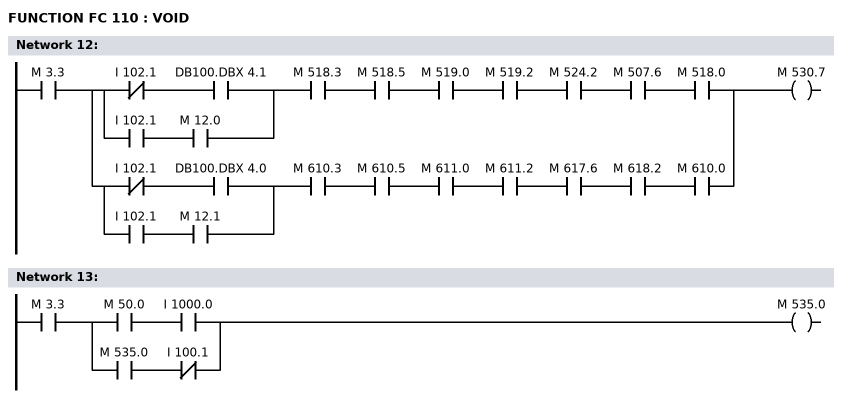

      A     M      3.3;
      A(    ;
      A(    ;
      AN    I    102.1;
      A     DB100.DBX    4.1;
      O     ;
      A     I    102.1;
      A     M     12.0;
      )     ;
      A     M    518.3;
      A     M    518.5;
      A     M    519.0;
      A     M    519.2;
      A     M    524.2;
      A     M    507.6;
      A     M    518.0;
      O     ;
      A(    ;
      AN    I    102.1;
      A     DB100.DBX    4.0;
      O     ;
      A     I    102.1;
      A     M     12.1;
      )     ;
      A     M    610.3;
      A     M    610.5;
      A     M    611.0;
      A     M    611.2;
      A     M    617.6;
      A     M    618.2;
      A     M    610.0;
      )     ;
      =     M    530.7;
NETWORK
TITLE =

      A     M      3.3;
      A(    ;
      A     M     50.0;
      A     I   1000.0;
      O     ;
      A     M    535.0;
      AN    I    100.1;
      )     ;
      =     M    535.0;
NETWORK
TITLE =

      AN    OV;
      =     L      0.0;
      A     L      0.0;
      A     I     32.2;
      =     M    540.0;
      A     L      0.0;
      AN    I     32.2;
      AN    I     32.3;
      AN    I     32.6;
      =     M    540.1;
      A     L      0.0;
      A     I     33.6;
      A     I     33.7;
      =     M    540.6;
      A     L      0.0;
      AN    I     33.6;
      AN    I     33.7;
      =     M    540.7;
NETWORK
TITLE =AUTO SIGNAL
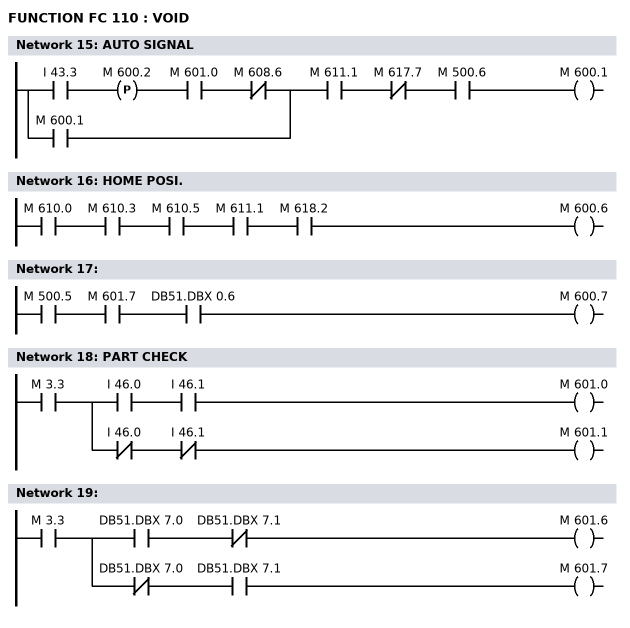

      A(    ;
      A     I     43.3;
      FP    M    600.2;
      A     M    601.0;
      AN    M    608.6;
      O     M    600.1;
      )     ;
      A     M    611.1;
      AN    M    617.7;
      A     M    500.6;
      =     M    600.1;
NETWORK
TITLE =HOME POSI.

      A     M    610.0;
      A     M    610.3;
      A     M    610.5;
      A     M    611.1;
      A     M    618.2;
      =     M    600.6;
NETWORK
TITLE =

      A     M    500.5;
      A     M    601.7;
      A     DB51.DBX    0.6;
      =     M    600.7;
NETWORK
TITLE =PART CHECK

      A     M      3.3;
      =     L      0.0;
      A     L      0.0;
      A     I     46.0;
      A     I     46.1;
      =     M    601.0;
      A     L      0.0;
      AN    I     46.0;
      AN    I     46.1;
      =     M    601.1;
NETWORK
TITLE =

      A     M      3.3;
      =     L      0.0;
      A     L      0.0;
      A     DB51.DBX    7.0;
      AN    DB51.DBX    7.1;
      =     M    601.6;
      A     L      0.0;
      AN    DB51.DBX    7.0;
      A     DB51.DBX    7.1;
      =     M    601.7;
END_FUNCTION

FUNCTION_BLOCK FB 111
TITLE =
VERSION : 0.1


VAR
  LM_PIN : FB 424;
  LM_CLAMP1 : FB 424;
  LM_CLAMP2 : FB 424;
  LM_SLIDE : FB 424;
  LM_SLIDE_ADV_LOCK : FB 424;
  LM_GUN1_SHIFT : FB 424;
  LM_GUN2_SHIFT : FB 424;
  LM_GUN2_LATCH : FB 424;
  TL_SLIDE : FB 424;
  TL_SLIDE_LOCK : FB 424;
  TL_PIN_UP_DOWN : FB 424;
  TL_CLAMP1_SOL : FB 424;
  TL_CLAMP2_SOL : FB 424;
  TL_GUN1_SHIFT : FB 424;
  TL_GUN2_SHIFT : FB 424;
  TL_GUN3_1_SHIFT : FB 424;
  TL_GUN3_2_SHIFT : FB 424;
  LM_IDLE_LATCH : FB 424;
  TL_IDLE_LATCH : FB 424;
  TL_IDLE_PIN : FB 424;
END_VAR
BEGIN
NETWORK
TITLE =
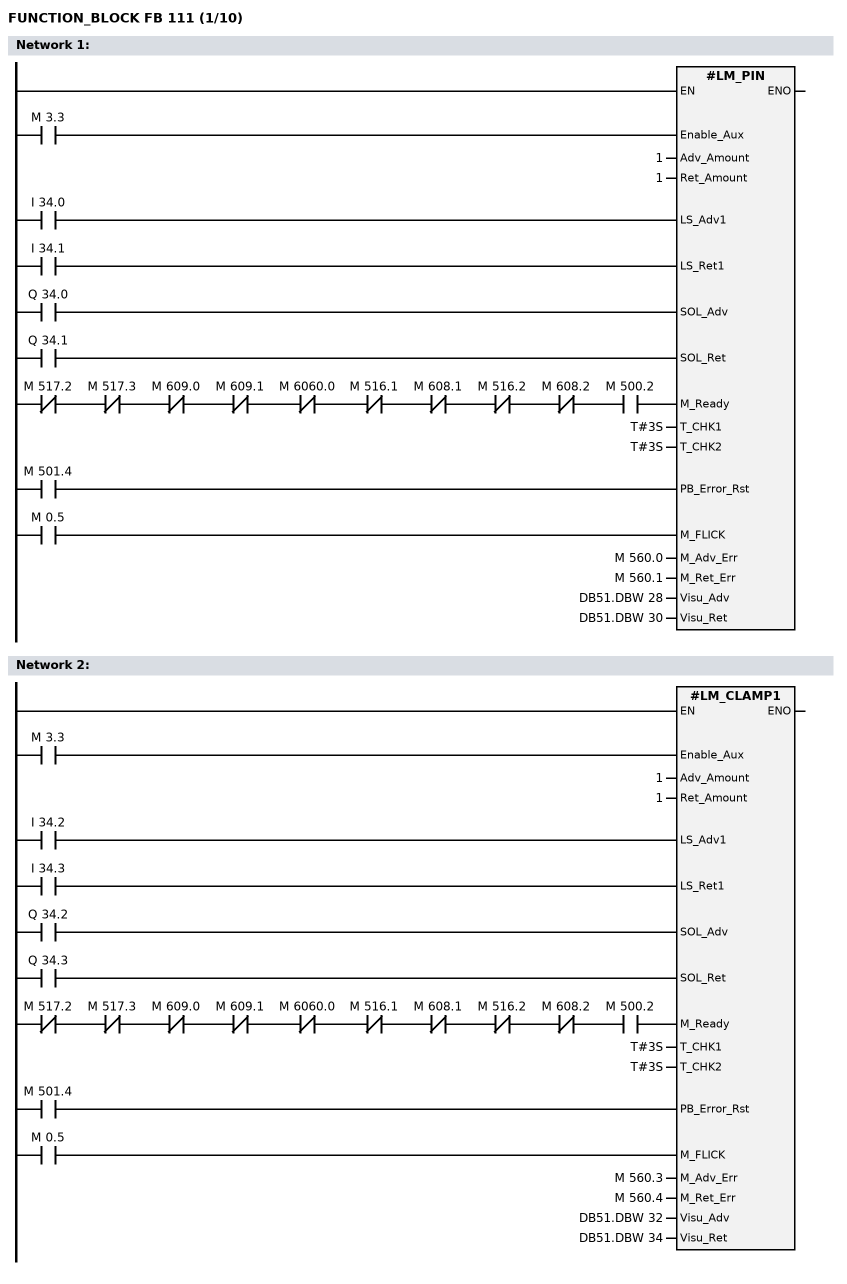

      A     M      3.3;
      =     L      0.0;
      BLD   103;
      A     I     34.0;
      =     L      0.1;
      BLD   103;
      A     I     34.1;
      =     L      0.2;
      BLD   103;
      A     Q     34.0;
      =     L      1.1;
      BLD   103;
      A     Q     34.1;
      =     L      1.2;
      BLD   103;
      AN    M    517.2;
      AN    M    517.3;
      AN    M    609.0;
      AN    M    609.1;
      AN    M   6060.0;
      AN    M    516.1;
      AN    M    608.1;
      AN    M    516.2;
      AN    M    608.2;
      A     M    500.2;
      =     L      1.3;
      BLD   103;
      A     M    501.4;
      =     L      1.5;
      BLD   103;
      A     M      0.5;
      =     L      1.6;
      BLD   103;
      CALL #LM_PIN (
           Enable_Aux               := L      0.0,
           Adv_Amount               := 1,
           Ret_Amount               := 1,
           LS_Adv1                  := L      0.1,
           LS_Ret1                  := L      0.2,
           SOL_Adv                  := L      1.1,
           SOL_Ret                  := L      1.2,
           M_Ready                  := L      1.3,
           T_CHK1                   := T#3S,
           T_CHK2                   := T#3S,
           PB_Error_Rst             := L      1.5,
           M_FLICK                  := L      1.6,
           M_Adv_Err                := M    560.0,
           M_Ret_Err                := M    560.1,
           Visu_Adv                 := DB51.DBW   28,
           Visu_Ret                 := DB51.DBW   30);
      NOP   0;
NETWORK
TITLE =

      A     M      3.3;
      =     L      0.0;
      BLD   103;
      A     I     34.2;
      =     L      0.1;
      BLD   103;
      A     I     34.3;
      =     L      0.2;
      BLD   103;
      A     Q     34.2;
      =     L      1.1;
      BLD   103;
      A     Q     34.3;
      =     L      1.2;
      BLD   103;
      AN    M    517.2;
      AN    M    517.3;
      AN    M    609.0;
      AN    M    609.1;
      AN    M   6060.0;
      AN    M    516.1;
      AN    M    608.1;
      AN    M    516.2;
      AN    M    608.2;
      A     M    500.2;
      =     L      1.3;
      BLD   103;
      A     M    501.4;
      =     L      1.5;
      BLD   103;
      A     M      0.5;
      =     L      1.6;
      BLD   103;
      CALL #LM_CLAMP1 (
           Enable_Aux               := L      0.0,
           Adv_Amount               := 1,
           Ret_Amount               := 1,
           LS_Adv1                  := L      0.1,
           LS_Ret1                  := L      0.2,
           SOL_Adv                  := L      1.1,
           SOL_Ret                  := L      1.2,
           M_Ready                  := L      1.3,
           T_CHK1                   := T#3S,
           T_CHK2                   := T#3S,
           PB_Error_Rst             := L      1.5,
           M_FLICK                  := L      1.6,
           M_Adv_Err                := M    560.3,
           M_Ret_Err                := M    560.4,
           Visu_Adv                 := DB51.DBW   32,
           Visu_Ret                 := DB51.DBW   34);
      NOP   0;
NETWORK
TITLE =
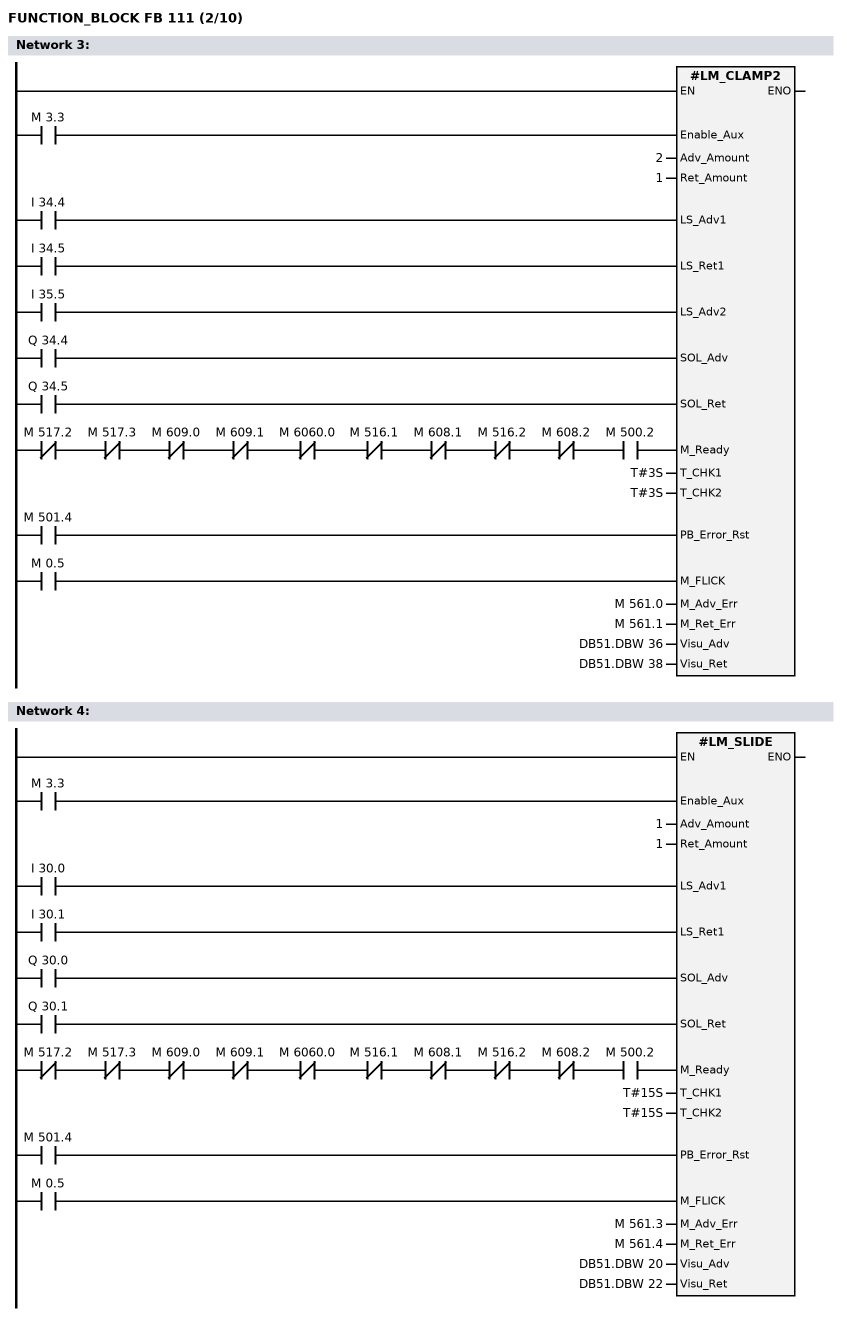

      A     M      3.3;
      =     L      0.0;
      BLD   103;
      A     I     34.4;
      =     L      0.1;
      BLD   103;
      A     I     34.5;
      =     L      0.2;
      BLD   103;
      A     I     35.5;
      =     L      0.3;
      BLD   103;
      A     Q     34.4;
      =     L      1.1;
      BLD   103;
      A     Q     34.5;
      =     L      1.2;
      BLD   103;
      AN    M    517.2;
      AN    M    517.3;
      AN    M    609.0;
      AN    M    609.1;
      AN    M   6060.0;
      AN    M    516.1;
      AN    M    608.1;
      AN    M    516.2;
      AN    M    608.2;
      A     M    500.2;
      =     L      1.3;
      BLD   103;
      A     M    501.4;
      =     L      1.5;
      BLD   103;
      A     M      0.5;
      =     L      1.6;
      BLD   103;
      CALL #LM_CLAMP2 (
           Enable_Aux               := L      0.0,
           Adv_Amount               := 2,
           Ret_Amount               := 1,
           LS_Adv1                  := L      0.1,
           LS_Ret1                  := L      0.2,
           LS_Adv2                  := L      0.3,
           SOL_Adv                  := L      1.1,
           SOL_Ret                  := L      1.2,
           M_Ready                  := L      1.3,
           T_CHK1                   := T#3S,
           T_CHK2                   := T#3S,
           PB_Error_Rst             := L      1.5,
           M_FLICK                  := L      1.6,
           M_Adv_Err                := M    561.0,
           M_Ret_Err                := M    561.1,
           Visu_Adv                 := DB51.DBW   36,
           Visu_Ret                 := DB51.DBW   38);
      NOP   0;
NETWORK
TITLE =

      A     M      3.3;
      =     L      0.0;
      BLD   103;
      A     I     30.0;
      =     L      0.1;
      BLD   103;
      A     I     30.1;
      =     L      0.2;
      BLD   103;
      A     Q     30.0;
      =     L      1.1;
      BLD   103;
      A     Q     30.1;
      =     L      1.2;
      BLD   103;
      AN    M    517.2;
      AN    M    517.3;
      AN    M    609.0;
      AN    M    609.1;
      AN    M   6060.0;
      AN    M    516.1;
      AN    M    608.1;
      AN    M    516.2;
      AN    M    608.2;
      A     M    500.2;
      =     L      1.3;
      BLD   103;
      A     M    501.4;
      =     L      1.5;
      BLD   103;
      A     M      0.5;
      =     L      1.6;
      BLD   103;
      CALL #LM_SLIDE (
           Enable_Aux               := L      0.0,
           Adv_Amount               := 1,
           Ret_Amount               := 1,
           LS_Adv1                  := L      0.1,
           LS_Ret1                  := L      0.2,
           SOL_Adv                  := L      1.1,
           SOL_Ret                  := L      1.2,
           M_Ready                  := L      1.3,
           T_CHK1                   := T#15S,
           T_CHK2                   := T#15S,
           PB_Error_Rst             := L      1.5,
           M_FLICK                  := L      1.6,
           M_Adv_Err                := M    561.3,
           M_Ret_Err                := M    561.4,
           Visu_Adv                 := DB51.DBW   20,
           Visu_Ret                 := DB51.DBW   22);
      NOP   0;
NETWORK
TITLE =
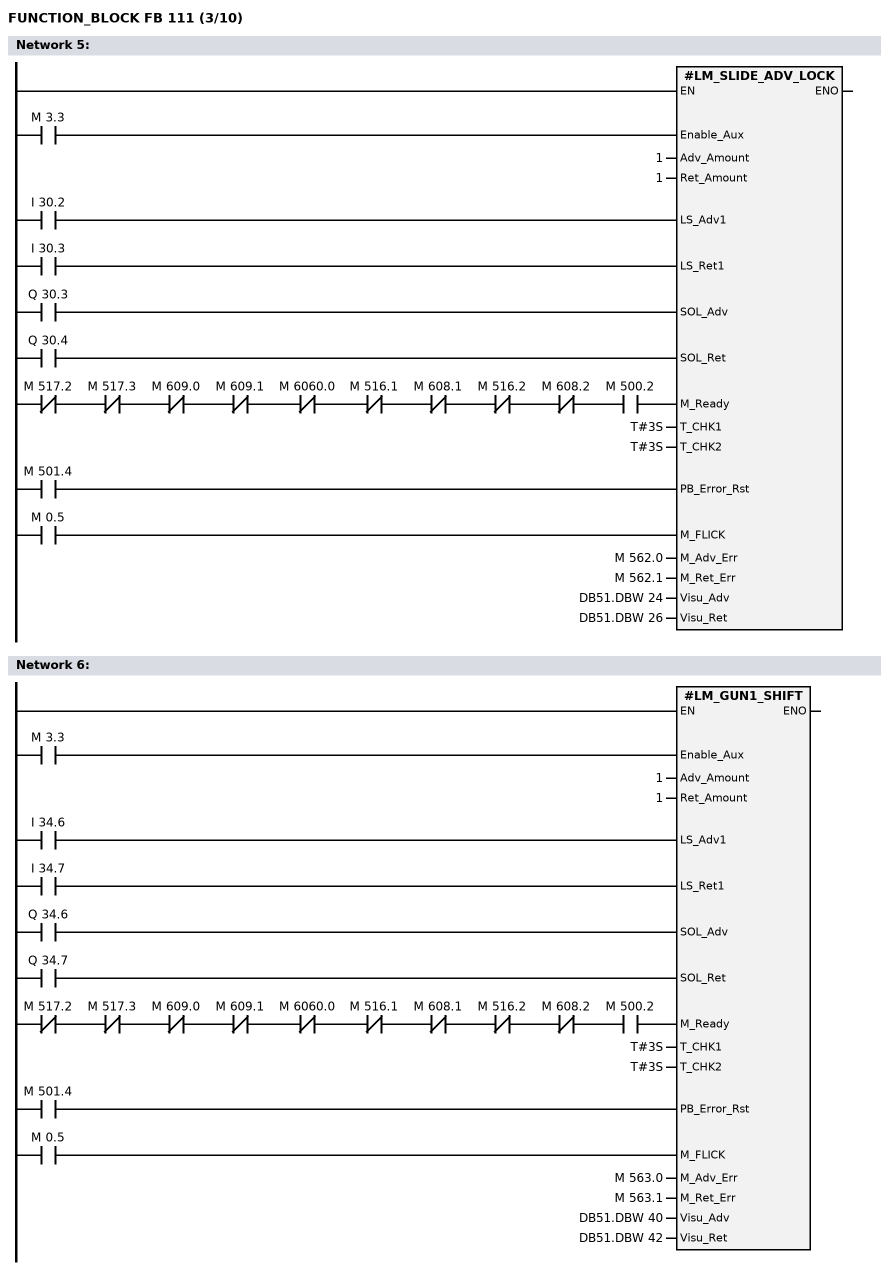

      A     M      3.3;
      =     L      0.0;
      BLD   103;
      A     I     30.2;
      =     L      0.1;
      BLD   103;
      A     I     30.3;
      =     L      0.2;
      BLD   103;
      A     Q     30.3;
      =     L      1.1;
      BLD   103;
      A     Q     30.4;
      =     L      1.2;
      BLD   103;
      AN    M    517.2;
      AN    M    517.3;
      AN    M    609.0;
      AN    M    609.1;
      AN    M   6060.0;
      AN    M    516.1;
      AN    M    608.1;
      AN    M    516.2;
      AN    M    608.2;
      A     M    500.2;
      =     L      1.3;
      BLD   103;
      A     M    501.4;
      =     L      1.5;
      BLD   103;
      A     M      0.5;
      =     L      1.6;
      BLD   103;
      CALL #LM_SLIDE_ADV_LOCK (
           Enable_Aux               := L      0.0,
           Adv_Amount               := 1,
           Ret_Amount               := 1,
           LS_Adv1                  := L      0.1,
           LS_Ret1                  := L      0.2,
           SOL_Adv                  := L      1.1,
           SOL_Ret                  := L      1.2,
           M_Ready                  := L      1.3,
           T_CHK1                   := T#3S,
           T_CHK2                   := T#3S,
           PB_Error_Rst             := L      1.5,
           M_FLICK                  := L      1.6,
           M_Adv_Err                := M    562.0,
           M_Ret_Err                := M    562.1,
           Visu_Adv                 := DB51.DBW   24,
           Visu_Ret                 := DB51.DBW   26);
      NOP   0;
NETWORK
TITLE =

      A     M      3.3;
      =     L      0.0;
      BLD   103;
      A     I     34.6;
      =     L      0.1;
      BLD   103;
      A     I     34.7;
      =     L      0.2;
      BLD   103;
      A     Q     34.6;
      =     L      1.1;
      BLD   103;
      A     Q     34.7;
      =     L      1.2;
      BLD   103;
      AN    M    517.2;
      AN    M    517.3;
      AN    M    609.0;
      AN    M    609.1;
      AN    M   6060.0;
      AN    M    516.1;
      AN    M    608.1;
      AN    M    516.2;
      AN    M    608.2;
      A     M    500.2;
      =     L      1.3;
      BLD   103;
      A     M    501.4;
      =     L      1.5;
      BLD   103;
      A     M      0.5;
      =     L      1.6;
      BLD   103;
      CALL #LM_GUN1_SHIFT (
           Enable_Aux               := L      0.0,
           Adv_Amount               := 1,
           Ret_Amount               := 1,
           LS_Adv1                  := L      0.1,
           LS_Ret1                  := L      0.2,
           SOL_Adv                  := L      1.1,
           SOL_Ret                  := L      1.2,
           M_Ready                  := L      1.3,
           T_CHK1                   := T#3S,
           T_CHK2                   := T#3S,
           PB_Error_Rst             := L      1.5,
           M_FLICK                  := L      1.6,
           M_Adv_Err                := M    563.0,
           M_Ret_Err                := M    563.1,
           Visu_Adv                 := DB51.DBW   40,
           Visu_Ret                 := DB51.DBW   42);
      NOP   0;
NETWORK
TITLE =
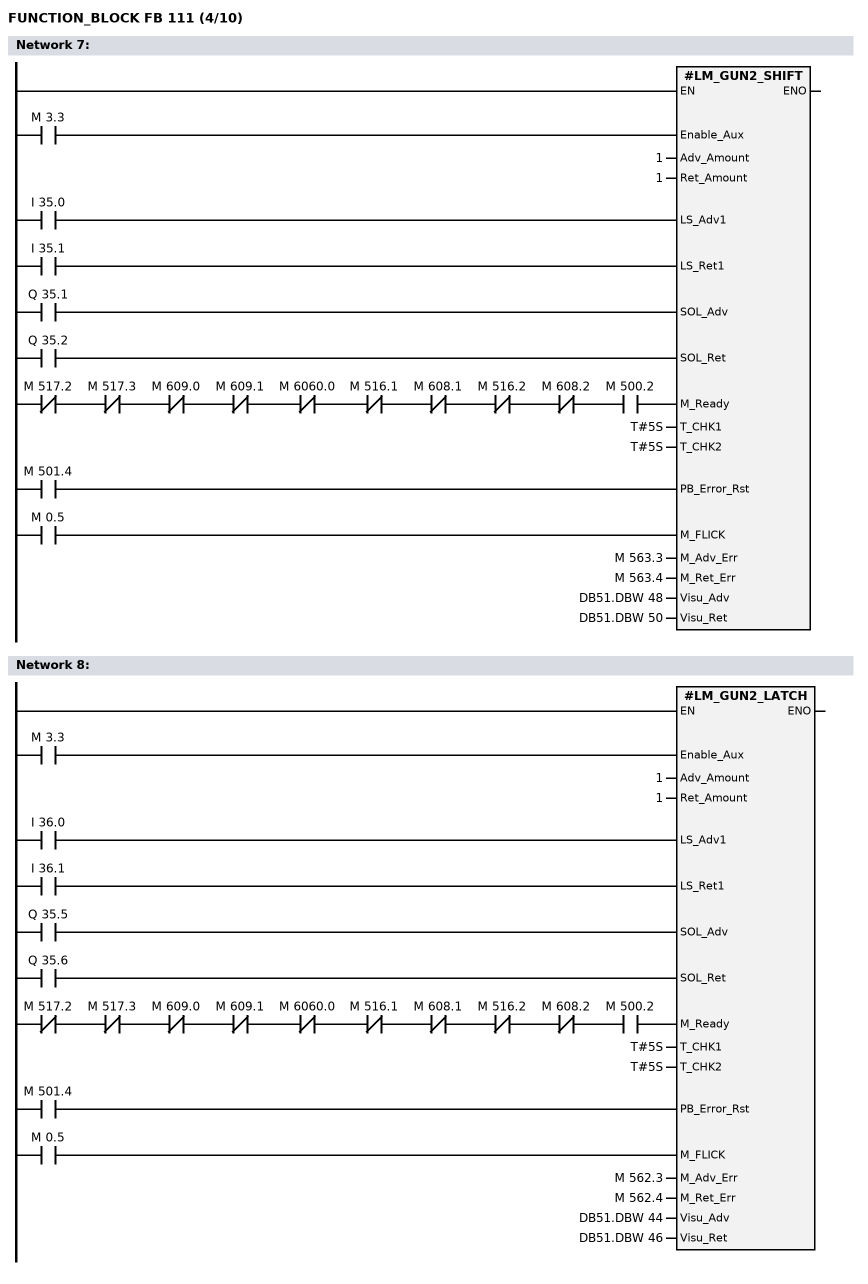

      A     M      3.3;
      =     L      0.0;
      BLD   103;
      A     I     35.0;
      =     L      0.1;
      BLD   103;
      A     I     35.1;
      =     L      0.2;
      BLD   103;
      A     Q     35.1;
      =     L      1.1;
      BLD   103;
      A     Q     35.2;
      =     L      1.2;
      BLD   103;
      AN    M    517.2;
      AN    M    517.3;
      AN    M    609.0;
      AN    M    609.1;
      AN    M   6060.0;
      AN    M    516.1;
      AN    M    608.1;
      AN    M    516.2;
      AN    M    608.2;
      A     M    500.2;
      =     L      1.3;
      BLD   103;
      A     M    501.4;
      =     L      1.5;
      BLD   103;
      A     M      0.5;
      =     L      1.6;
      BLD   103;
      CALL #LM_GUN2_SHIFT (
           Enable_Aux               := L      0.0,
           Adv_Amount               := 1,
           Ret_Amount               := 1,
           LS_Adv1                  := L      0.1,
           LS_Ret1                  := L      0.2,
           SOL_Adv                  := L      1.1,
           SOL_Ret                  := L      1.2,
           M_Ready                  := L      1.3,
           T_CHK1                   := T#5S,
           T_CHK2                   := T#5S,
           PB_Error_Rst             := L      1.5,
           M_FLICK                  := L      1.6,
           M_Adv_Err                := M    563.3,
           M_Ret_Err                := M    563.4,
           Visu_Adv                 := DB51.DBW   48,
           Visu_Ret                 := DB51.DBW   50);
      NOP   0;
NETWORK
TITLE =

      A     M      3.3;
      =     L      0.0;
      BLD   103;
      A     I     36.0;
      =     L      0.1;
      BLD   103;
      A     I     36.1;
      =     L      0.2;
      BLD   103;
      A     Q     35.5;
      =     L      1.1;
      BLD   103;
      A     Q     35.6;
      =     L      1.2;
      BLD   103;
      AN    M    517.2;
      AN    M    517.3;
      AN    M    609.0;
      AN    M    609.1;
      AN    M   6060.0;
      AN    M    516.1;
      AN    M    608.1;
      AN    M    516.2;
      AN    M    608.2;
      A     M    500.2;
      =     L      1.3;
      BLD   103;
      A     M    501.4;
      =     L      1.5;
      BLD   103;
      A     M      0.5;
      =     L      1.6;
      BLD   103;
      CALL #LM_GUN2_LATCH (
           Enable_Aux               := L      0.0,
           Adv_Amount               := 1,
           Ret_Amount               := 1,
           LS_Adv1                  := L      0.1,
           LS_Ret1                  := L      0.2,
           SOL_Adv                  := L      1.1,
           SOL_Ret                  := L      1.2,
           M_Ready                  := L      1.3,
           T_CHK1                   := T#5S,
           T_CHK2                   := T#5S,
           PB_Error_Rst             := L      1.5,
           M_FLICK                  := L      1.6,
           M_Adv_Err                := M    562.3,
           M_Ret_Err                := M    562.4,
           Visu_Adv                 := DB51.DBW   44,
           Visu_Ret                 := DB51.DBW   46);
      NOP   0;
NETWORK
TITLE =
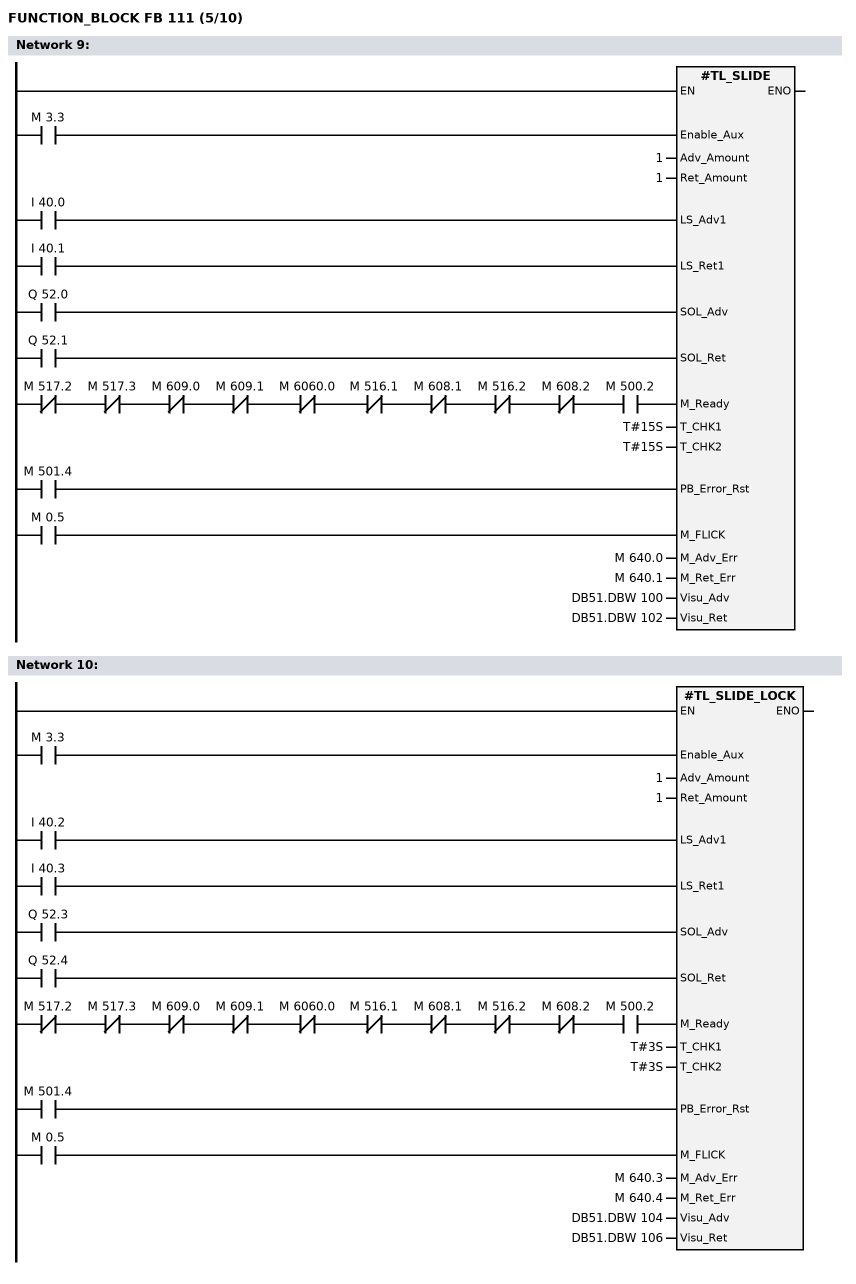

      A     M      3.3;
      =     L      0.0;
      BLD   103;
      A     I     40.0;
      =     L      0.1;
      BLD   103;
      A     I     40.1;
      =     L      0.2;
      BLD   103;
      A     Q     52.0;
      =     L      1.1;
      BLD   103;
      A     Q     52.1;
      =     L      1.2;
      BLD   103;
      AN    M    517.2;
      AN    M    517.3;
      AN    M    609.0;
      AN    M    609.1;
      AN    M   6060.0;
      AN    M    516.1;
      AN    M    608.1;
      AN    M    516.2;
      AN    M    608.2;
      A     M    500.2;
      =     L      1.3;
      BLD   103;
      A     M    501.4;
      =     L      1.5;
      BLD   103;
      A     M      0.5;
      =     L      1.6;
      BLD   103;
      CALL #TL_SLIDE (
           Enable_Aux               := L      0.0,
           Adv_Amount               := 1,
           Ret_Amount               := 1,
           LS_Adv1                  := L      0.1,
           LS_Ret1                  := L      0.2,
           SOL_Adv                  := L      1.1,
           SOL_Ret                  := L      1.2,
           M_Ready                  := L      1.3,
           T_CHK1                   := T#15S,
           T_CHK2                   := T#15S,
           PB_Error_Rst             := L      1.5,
           M_FLICK                  := L      1.6,
           M_Adv_Err                := M    640.0,
           M_Ret_Err                := M    640.1,
           Visu_Adv                 := DB51.DBW  100,
           Visu_Ret                 := DB51.DBW  102);
      NOP   0;
NETWORK
TITLE =

      A     M      3.3;
      =     L      0.0;
      BLD   103;
      A     I     40.2;
      =     L      0.1;
      BLD   103;
      A     I     40.3;
      =     L      0.2;
      BLD   103;
      A     Q     52.3;
      =     L      1.1;
      BLD   103;
      A     Q     52.4;
      =     L      1.2;
      BLD   103;
      AN    M    517.2;
      AN    M    517.3;
      AN    M    609.0;
      AN    M    609.1;
      AN    M   6060.0;
      AN    M    516.1;
      AN    M    608.1;
      AN    M    516.2;
      AN    M    608.2;
      A     M    500.2;
      =     L      1.3;
      BLD   103;
      A     M    501.4;
      =     L      1.5;
      BLD   103;
      A     M      0.5;
      =     L      1.6;
      BLD   103;
      CALL #TL_SLIDE_LOCK (
           Enable_Aux               := L      0.0,
           Adv_Amount               := 1,
           Ret_Amount               := 1,
           LS_Adv1                  := L      0.1,
           LS_Ret1                  := L      0.2,
           SOL_Adv                  := L      1.1,
           SOL_Ret                  := L      1.2,
           M_Ready                  := L      1.3,
           T_CHK1                   := T#3S,
           T_CHK2                   := T#3S,
           PB_Error_Rst             := L      1.5,
           M_FLICK                  := L      1.6,
           M_Adv_Err                := M    640.3,
           M_Ret_Err                := M    640.4,
           Visu_Adv                 := DB51.DBW  104,
           Visu_Ret                 := DB51.DBW  106);
      NOP   0;
NETWORK
TITLE =
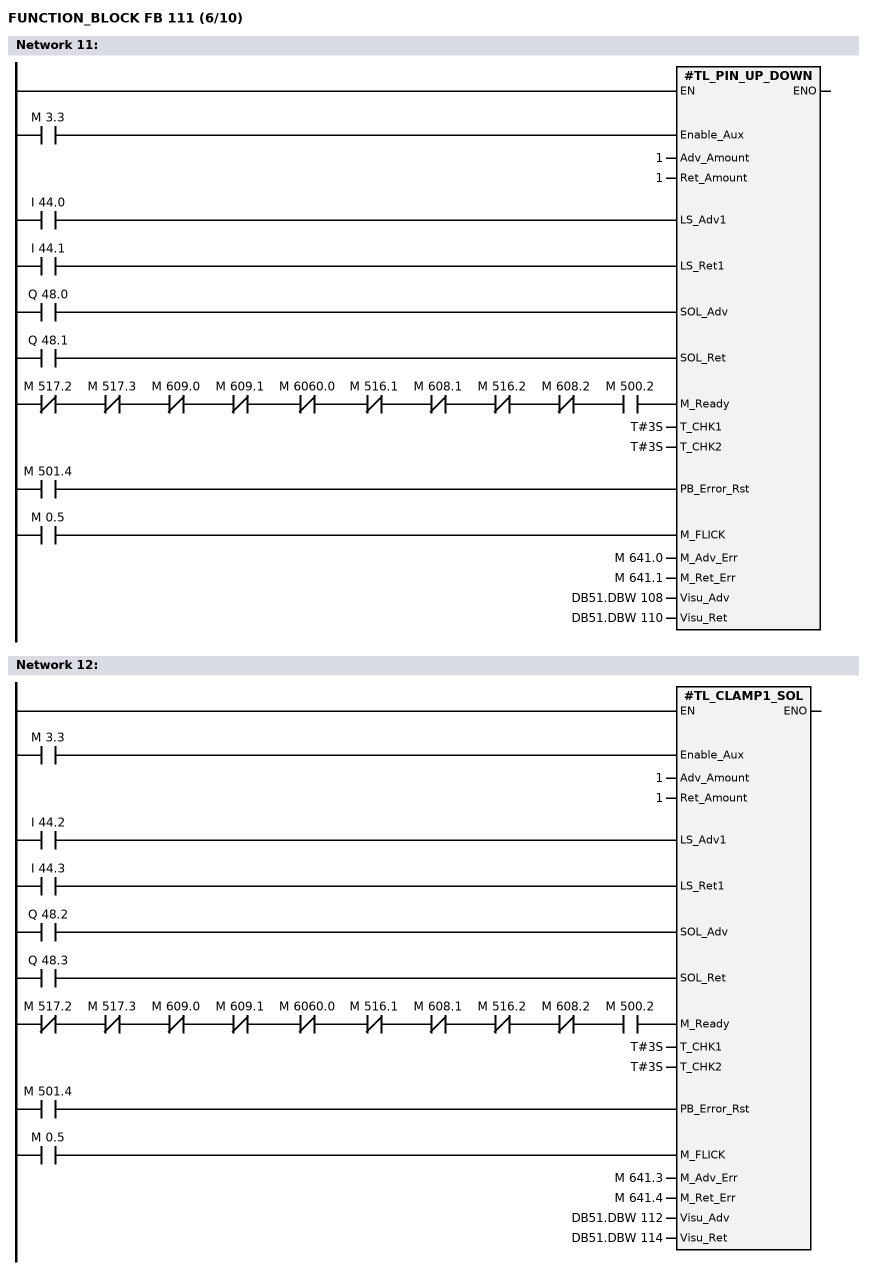

      A     M      3.3;
      =     L      0.0;
      BLD   103;
      A     I     44.0;
      =     L      0.1;
      BLD   103;
      A     I     44.1;
      =     L      0.2;
      BLD   103;
      A     Q     48.0;
      =     L      1.1;
      BLD   103;
      A     Q     48.1;
      =     L      1.2;
      BLD   103;
      AN    M    517.2;
      AN    M    517.3;
      AN    M    609.0;
      AN    M    609.1;
      AN    M   6060.0;
      AN    M    516.1;
      AN    M    608.1;
      AN    M    516.2;
      AN    M    608.2;
      A     M    500.2;
      =     L      1.3;
      BLD   103;
      A     M    501.4;
      =     L      1.5;
      BLD   103;
      A     M      0.5;
      =     L      1.6;
      BLD   103;
      CALL #TL_PIN_UP_DOWN (
           Enable_Aux               := L      0.0,
           Adv_Amount               := 1,
           Ret_Amount               := 1,
           LS_Adv1                  := L      0.1,
           LS_Ret1                  := L      0.2,
           SOL_Adv                  := L      1.1,
           SOL_Ret                  := L      1.2,
           M_Ready                  := L      1.3,
           T_CHK1                   := T#3S,
           T_CHK2                   := T#3S,
           PB_Error_Rst             := L      1.5,
           M_FLICK                  := L      1.6,
           M_Adv_Err                := M    641.0,
           M_Ret_Err                := M    641.1,
           Visu_Adv                 := DB51.DBW  108,
           Visu_Ret                 := DB51.DBW  110);
      NOP   0;
NETWORK
TITLE =

      A     M      3.3;
      =     L      0.0;
      BLD   103;
      A     I     44.2;
      =     L      0.1;
      BLD   103;
      A     I     44.3;
      =     L      0.2;
      BLD   103;
      A     Q     48.2;
      =     L      1.1;
      BLD   103;
      A     Q     48.3;
      =     L      1.2;
      BLD   103;
      AN    M    517.2;
      AN    M    517.3;
      AN    M    609.0;
      AN    M    609.1;
      AN    M   6060.0;
      AN    M    516.1;
      AN    M    608.1;
      AN    M    516.2;
      AN    M    608.2;
      A     M    500.2;
      =     L      1.3;
      BLD   103;
      A     M    501.4;
      =     L      1.5;
      BLD   103;
      A     M      0.5;
      =     L      1.6;
      BLD   103;
      CALL #TL_CLAMP1_SOL (
           Enable_Aux               := L      0.0,
           Adv_Amount               := 1,
           Ret_Amount               := 1,
           LS_Adv1                  := L      0.1,
           LS_Ret1                  := L      0.2,
           SOL_Adv                  := L      1.1,
           SOL_Ret                  := L      1.2,
           M_Ready                  := L      1.3,
           T_CHK1                   := T#3S,
           T_CHK2                   := T#3S,
           PB_Error_Rst             := L      1.5,
           M_FLICK                  := L      1.6,
           M_Adv_Err                := M    641.3,
           M_Ret_Err                := M    641.4,
           Visu_Adv                 := DB51.DBW  112,
           Visu_Ret                 := DB51.DBW  114);
      NOP   0;
NETWORK
TITLE =
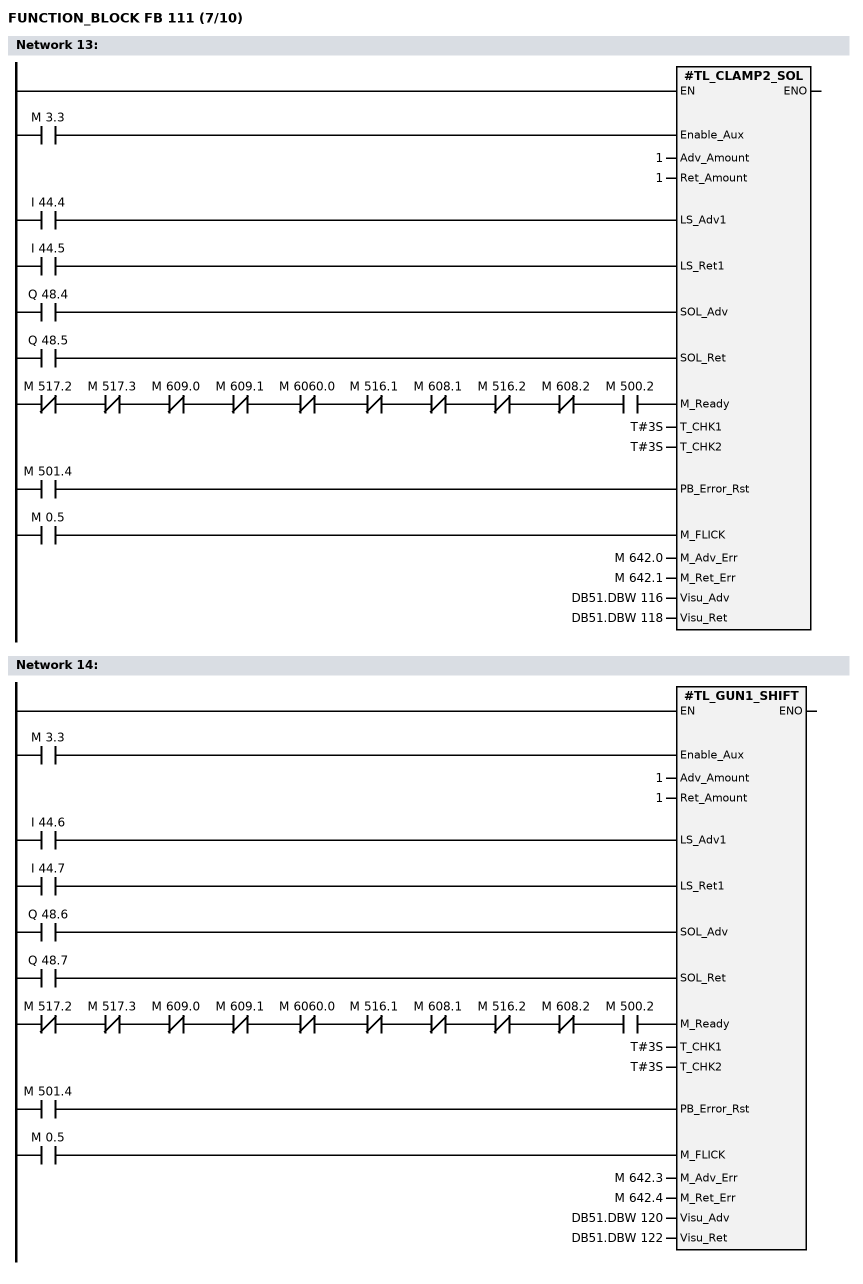

      A     M      3.3;
      =     L      0.0;
      BLD   103;
      A     I     44.4;
      =     L      0.1;
      BLD   103;
      A     I     44.5;
      =     L      0.2;
      BLD   103;
      A     Q     48.4;
      =     L      1.1;
      BLD   103;
      A     Q     48.5;
      =     L      1.2;
      BLD   103;
      AN    M    517.2;
      AN    M    517.3;
      AN    M    609.0;
      AN    M    609.1;
      AN    M   6060.0;
      AN    M    516.1;
      AN    M    608.1;
      AN    M    516.2;
      AN    M    608.2;
      A     M    500.2;
      =     L      1.3;
      BLD   103;
      A     M    501.4;
      =     L      1.5;
      BLD   103;
      A     M      0.5;
      =     L      1.6;
      BLD   103;
      CALL #TL_CLAMP2_SOL (
           Enable_Aux               := L      0.0,
           Adv_Amount               := 1,
           Ret_Amount               := 1,
           LS_Adv1                  := L      0.1,
           LS_Ret1                  := L      0.2,
           SOL_Adv                  := L      1.1,
           SOL_Ret                  := L      1.2,
           M_Ready                  := L      1.3,
           T_CHK1                   := T#3S,
           T_CHK2                   := T#3S,
           PB_Error_Rst             := L      1.5,
           M_FLICK                  := L      1.6,
           M_Adv_Err                := M    642.0,
           M_Ret_Err                := M    642.1,
           Visu_Adv                 := DB51.DBW  116,
           Visu_Ret                 := DB51.DBW  118);
      NOP   0;
NETWORK
TITLE =

      A     M      3.3;
      =     L      0.0;
      BLD   103;
      A     I     44.6;
      =     L      0.1;
      BLD   103;
      A     I     44.7;
      =     L      0.2;
      BLD   103;
      A     Q     48.6;
      =     L      1.1;
      BLD   103;
      A     Q     48.7;
      =     L      1.2;
      BLD   103;
      AN    M    517.2;
      AN    M    517.3;
      AN    M    609.0;
      AN    M    609.1;
      AN    M   6060.0;
      AN    M    516.1;
      AN    M    608.1;
      AN    M    516.2;
      AN    M    608.2;
      A     M    500.2;
      =     L      1.3;
      BLD   103;
      A     M    501.4;
      =     L      1.5;
      BLD   103;
      A     M      0.5;
      =     L      1.6;
      BLD   103;
      CALL #TL_GUN1_SHIFT (
           Enable_Aux               := L      0.0,
           Adv_Amount               := 1,
           Ret_Amount               := 1,
           LS_Adv1                  := L      0.1,
           LS_Ret1                  := L      0.2,
           SOL_Adv                  := L      1.1,
           SOL_Ret                  := L      1.2,
           M_Ready                  := L      1.3,
           T_CHK1                   := T#3S,
           T_CHK2                   := T#3S,
           PB_Error_Rst             := L      1.5,
           M_FLICK                  := L      1.6,
           M_Adv_Err                := M    642.3,
           M_Ret_Err                := M    642.4,
           Visu_Adv                 := DB51.DBW  120,
           Visu_Ret                 := DB51.DBW  122);
      NOP   0;
NETWORK
TITLE =
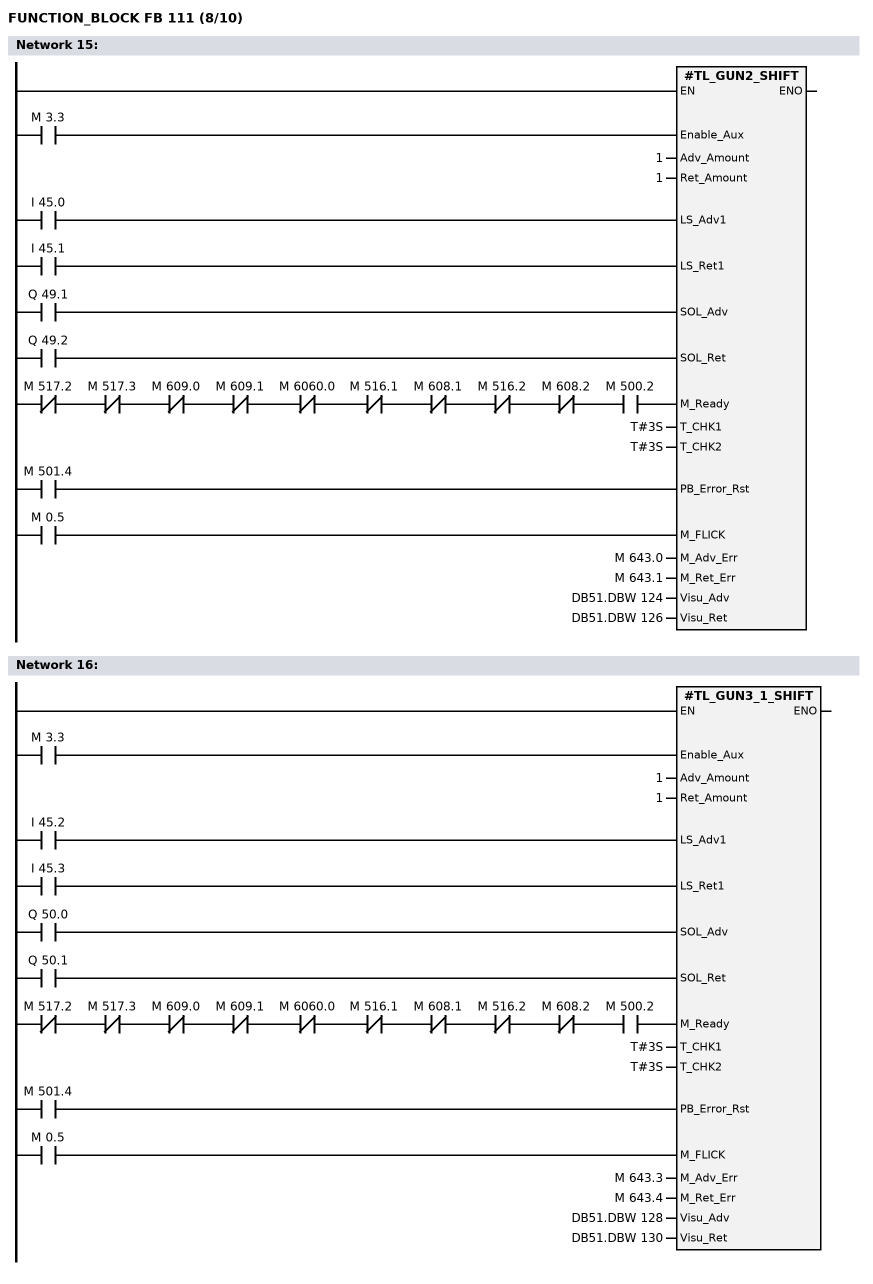

      A     M      3.3;
      =     L      0.0;
      BLD   103;
      A     I     45.0;
      =     L      0.1;
      BLD   103;
      A     I     45.1;
      =     L      0.2;
      BLD   103;
      A     Q     49.1;
      =     L      1.1;
      BLD   103;
      A     Q     49.2;
      =     L      1.2;
      BLD   103;
      AN    M    517.2;
      AN    M    517.3;
      AN    M    609.0;
      AN    M    609.1;
      AN    M   6060.0;
      AN    M    516.1;
      AN    M    608.1;
      AN    M    516.2;
      AN    M    608.2;
      A     M    500.2;
      =     L      1.3;
      BLD   103;
      A     M    501.4;
      =     L      1.5;
      BLD   103;
      A     M      0.5;
      =     L      1.6;
      BLD   103;
      CALL #TL_GUN2_SHIFT (
           Enable_Aux               := L      0.0,
           Adv_Amount               := 1,
           Ret_Amount               := 1,
           LS_Adv1                  := L      0.1,
           LS_Ret1                  := L      0.2,
           SOL_Adv                  := L      1.1,
           SOL_Ret                  := L      1.2,
           M_Ready                  := L      1.3,
           T_CHK1                   := T#3S,
           T_CHK2                   := T#3S,
           PB_Error_Rst             := L      1.5,
           M_FLICK                  := L      1.6,
           M_Adv_Err                := M    643.0,
           M_Ret_Err                := M    643.1,
           Visu_Adv                 := DB51.DBW  124,
           Visu_Ret                 := DB51.DBW  126);
      NOP   0;
NETWORK
TITLE =

      A     M      3.3;
      =     L      0.0;
      BLD   103;
      A     I     45.2;
      =     L      0.1;
      BLD   103;
      A     I     45.3;
      =     L      0.2;
      BLD   103;
      A     Q     50.0;
      =     L      1.1;
      BLD   103;
      A     Q     50.1;
      =     L      1.2;
      BLD   103;
      AN    M    517.2;
      AN    M    517.3;
      AN    M    609.0;
      AN    M    609.1;
      AN    M   6060.0;
      AN    M    516.1;
      AN    M    608.1;
      AN    M    516.2;
      AN    M    608.2;
      A     M    500.2;
      =     L      1.3;
      BLD   103;
      A     M    501.4;
      =     L      1.5;
      BLD   103;
      A     M      0.5;
      =     L      1.6;
      BLD   103;
      CALL #TL_GUN3_1_SHIFT (
           Enable_Aux               := L      0.0,
           Adv_Amount               := 1,
           Ret_Amount               := 1,
           LS_Adv1                  := L      0.1,
           LS_Ret1                  := L      0.2,
           SOL_Adv                  := L      1.1,
           SOL_Ret                  := L      1.2,
           M_Ready                  := L      1.3,
           T_CHK1                   := T#3S,
           T_CHK2                   := T#3S,
           PB_Error_Rst             := L      1.5,
           M_FLICK                  := L      1.6,
           M_Adv_Err                := M    643.3,
           M_Ret_Err                := M    643.4,
           Visu_Adv                 := DB51.DBW  128,
           Visu_Ret                 := DB51.DBW  130);
      NOP   0;
NETWORK
TITLE =
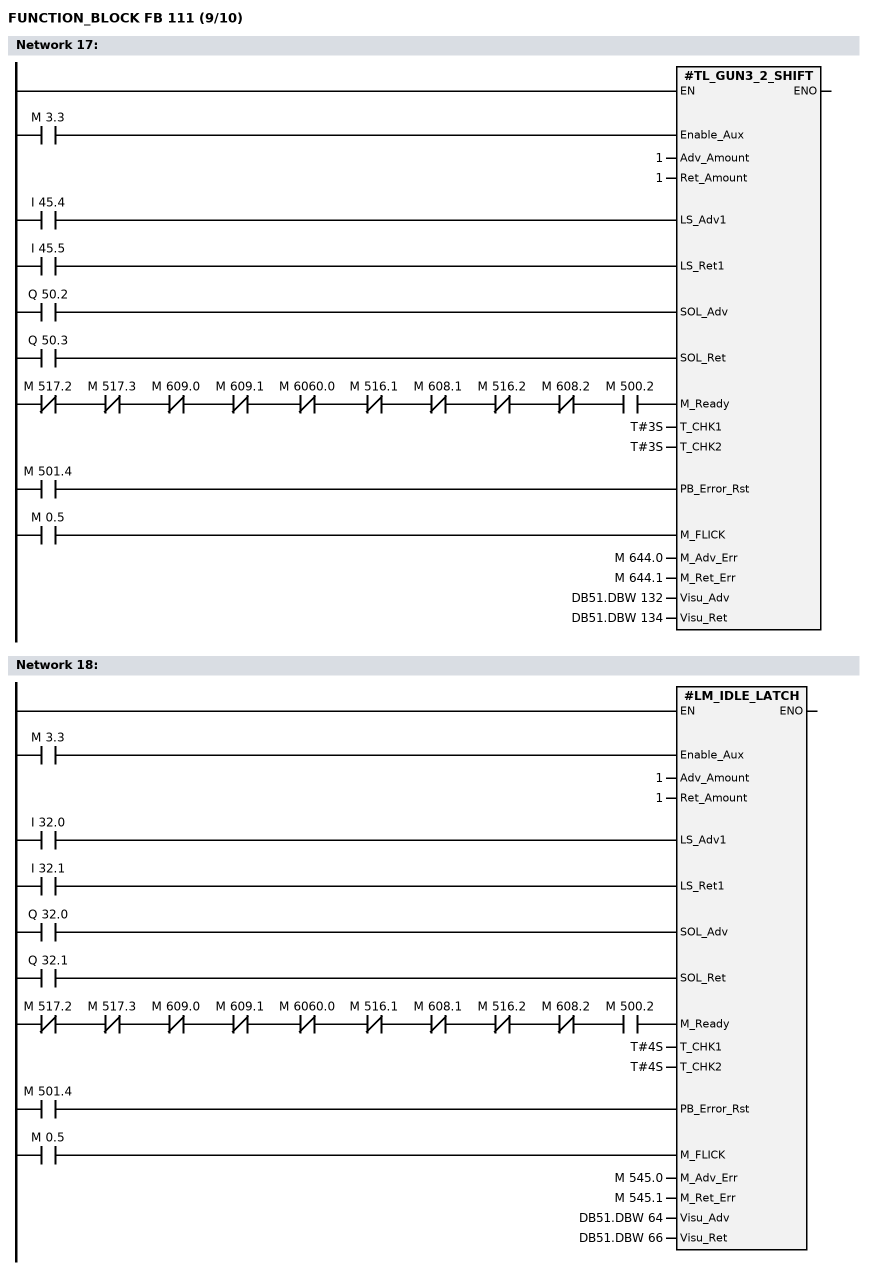

      A     M      3.3;
      =     L      0.0;
      BLD   103;
      A     I     45.4;
      =     L      0.1;
      BLD   103;
      A     I     45.5;
      =     L      0.2;
      BLD   103;
      A     Q     50.2;
      =     L      1.1;
      BLD   103;
      A     Q     50.3;
      =     L      1.2;
      BLD   103;
      AN    M    517.2;
      AN    M    517.3;
      AN    M    609.0;
      AN    M    609.1;
      AN    M   6060.0;
      AN    M    516.1;
      AN    M    608.1;
      AN    M    516.2;
      AN    M    608.2;
      A     M    500.2;
      =     L      1.3;
      BLD   103;
      A     M    501.4;
      =     L      1.5;
      BLD   103;
      A     M      0.5;
      =     L      1.6;
      BLD   103;
      CALL #TL_GUN3_2_SHIFT (
           Enable_Aux               := L      0.0,
           Adv_Amount               := 1,
           Ret_Amount               := 1,
           LS_Adv1                  := L      0.1,
           LS_Ret1                  := L      0.2,
           SOL_Adv                  := L      1.1,
           SOL_Ret                  := L      1.2,
           M_Ready                  := L      1.3,
           T_CHK1                   := T#3S,
           T_CHK2                   := T#3S,
           PB_Error_Rst             := L      1.5,
           M_FLICK                  := L      1.6,
           M_Adv_Err                := M    644.0,
           M_Ret_Err                := M    644.1,
           Visu_Adv                 := DB51.DBW  132,
           Visu_Ret                 := DB51.DBW  134);
      NOP   0;
NETWORK
TITLE =

      A     M      3.3;
      =     L      0.0;
      BLD   103;
      A     I     32.0;
      =     L      0.1;
      BLD   103;
      A     I     32.1;
      =     L      0.2;
      BLD   103;
      A     Q     32.0;
      =     L      1.1;
      BLD   103;
      A     Q     32.1;
      =     L      1.2;
      BLD   103;
      AN    M    517.2;
      AN    M    517.3;
      AN    M    609.0;
      AN    M    609.1;
      AN    M   6060.0;
      AN    M    516.1;
      AN    M    608.1;
      AN    M    516.2;
      AN    M    608.2;
      A     M    500.2;
      =     L      1.3;
      BLD   103;
      A     M    501.4;
      =     L      1.5;
      BLD   103;
      A     M      0.5;
      =     L      1.6;
      BLD   103;
      CALL #LM_IDLE_LATCH (
           Enable_Aux               := L      0.0,
           Adv_Amount               := 1,
           Ret_Amount               := 1,
           LS_Adv1                  := L      0.1,
           LS_Ret1                  := L      0.2,
           SOL_Adv                  := L      1.1,
           SOL_Ret                  := L      1.2,
           M_Ready                  := L      1.3,
           T_CHK1                   := T#4S,
           T_CHK2                   := T#4S,
           PB_Error_Rst             := L      1.5,
           M_FLICK                  := L      1.6,
           M_Adv_Err                := M    545.0,
           M_Ret_Err                := M    545.1,
           Visu_Adv                 := DB51.DBW   64,
           Visu_Ret                 := DB51.DBW   66);
      NOP   0;
NETWORK
TITLE =
